KUKA KRL program: MyProgram_013().src

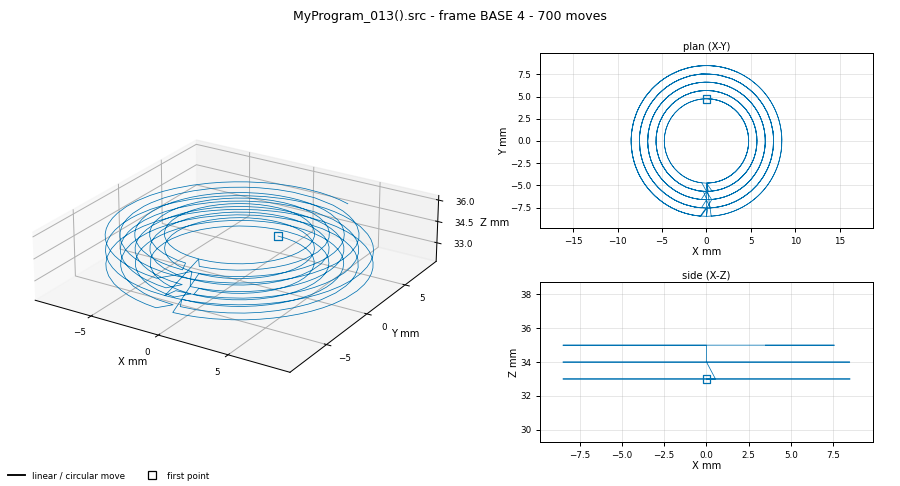
[picture p0: tool path of MyProgram_013().src in frame BASE 4, 700 of 700 moves have a stored position in this frame; points joined in program order, loops and branches not executed]
&ACCESS RVP
&REL 1
&PARAM TEMPLATE = C:\KRC\Roboter\Template\vorgabe
&PARAM EDITMASK = *
DEF MyProgram_013()
; ---- Setting reference (Base) ----
$BASE = BASE_DATA[4]

; --------------------------
; ---- Setting tool (TCP) ----
$TOOL = TOOL_DATA[3]
; --------------------------

$VEL.CP = VEL_APROX_PRINT
Startdeposition()
$VEL.CP = VEL_PRINT
LIN {X -0.0007,Y 4.7501,Z 33,A -2.5066,B 0,C 0,E1 0.1598,E2 90.0722} C_DIS
LIN {X 0.6681,Y 4.7058,Z 33,A -2.4838,B 0,C 0,E1 0.1598,E2 90.0722} C_DIS
LIN {X 1.3234,Y 4.564,Z 33,A -2.4657,B 0,C 0,E1 0.1598,E2 90.0722} C_DIS
LIN {X 1.9517,Y 4.3306,Z 33,A -2.4524,B 0,C 0,E1 0.1598,E2 90.0722} C_DIS
LIN {X 2.5415,Y 4.0125,Z 33,A -2.4441,B 0,C 0,E1 0.1598,E2 90.0722} C_DIS
LIN {X 3.0824,Y 3.6166,Z 33,A -2.441,B 0,C 0,E1 0.1598,E2 90.0722} C_DIS
LIN {X 3.561,Y 3.1471,Z 33,A -2.4432,B 0,C 0,E1 0.1598,E2 90.0722} C_DIS
LIN {X 3.9664,Y 2.6132,Z 33,A -2.4509,B 0,C 0,E1 0.1598,E2 90.0722} C_DIS
LIN {X 4.2946,Y 2.0289,Z 33,A -2.4637,B 0,C 0,E1 0.1598,E2 90.0721} C_DIS
LIN {X 4.5387,Y 1.4047,Z 33,A -2.4812,B 0,C 0,E1 0.1598,E2 90.0721} C_DIS
LIN {X 4.6913,Y 0.7521,Z 33,A -2.5033,B 0,C 0,E1 0.1598,E2 90.072} C_DIS
LIN {X 4.7501,Y 0.0845,Z 33,A -2.5295,B 0,C 0,E1 0.1598,E2 90.072} C_DIS
LIN {X 4.7153,Y -0.5848,Z 33,A -2.5593,B 0,C 0,E1 0.1598,E2 90.072} C_DIS
LIN {X 4.5852,Y -1.2423,Z 33,A -2.592,B 0,C 0,E1 0.1598,E2 90.0719} C_DIS
LIN {X 4.3645,Y -1.8751,Z 33,A -2.6271,B 0,C 0,E1 0.1598,E2 90.0719} C_DIS
LIN {X 4.0581,Y -2.4712,Z 33,A -2.6637,B 0,C 0,E1 0.1598,E2 90.0719} C_DIS
LIN {X 3.6691,Y -3.0171,Z 33,A -2.7013,B 0,C 0,E1 0.1598,E2 90.0719} C_DIS
LIN {X 3.2075,Y -3.5028,Z 33,A -2.7389,B 0,C 0,E1 0.1598,E2 90.0719} C_DIS
LIN {X 2.6831,Y -3.9201,Z 33,A -2.776,B 0,C 0,E1 0.1598,E2 90.0718} C_DIS
LIN {X 2.1055,Y -4.2604,Z 33,A -2.8117,B 0,C 0,E1 0.1598,E2 90.0718} C_DIS
LIN {X 1.4851,Y -4.5147,Z 33,A -2.8453,B 0,C 0,E1 0.1598,E2 90.0718} C_DIS
LIN {X 0.8351,Y -4.6789,Z 33,A -2.8762,B 0,C 0,E1 0.1598,E2 90.0718} C_DIS
LIN {X 0.0007,Y -4.7531,Z 33,A -2.9099,B 0,C 0,E1 0.1598,E2 90.0717} C_DIS
Enddeposition()
LIN {X 0.0007,Y -4.7531,Z 33,A -2.9099,B 0,C 0,E1 0.1598,E2 90.0717} C_DIS
Startdeposition()
$VEL.CP = VEL_PRINT
LIN {X 0.2137,Y -5.6787,Z 33,A -2.941,B 0,C 0,E1 0.1598,E2 90.0711} C_DIS
LIN {X 1.0439,Y -5.585,Z 33,A -2.9071,B 0,C 0,E1 0.1598,E2 90.0717} C_DIS
LIN {X 1.8527,Y -5.375,Z 33,A -2.8685,B 0,C 0,E1 0.1598,E2 90.0717} C_DIS
LIN {X 2.6206,Y -5.0447,Z 33,A -2.8262,B 0,C 0,E1 0.1598,E2 90.0717} C_DIS
LIN {X 3.3323,Y -4.6064,Z 33,A -2.7814,B 0,C 0,E1 0.1598,E2 90.0717} C_DIS
LIN {X 3.9709,Y -4.067,Z 33,A -2.735,B 0,C 0,E1 0.1598,E2 90.0717} C_DIS
LIN {X 4.5249,Y -3.4414,Z 33,A -2.6879,B 0,C 0,E1 0.1598,E2 90.0717} C_DIS
LIN {X 4.9785,Y -2.7397,Z 33,A -2.6413,B 0,C 0,E1 0.1598,E2 90.0717} C_DIS
LIN {X 5.3268,Y -1.9802,Z 33,A -2.5962,B 0,C 0,E1 0.1598,E2 90.0717} C_DIS
LIN {X 5.5609,Y -1.178,Z 33,A -2.5534,B 0,C 0,E1 0.1598,E2 90.0718} C_DIS
LIN {X 5.6744,Y -0.3499,Z 33,A -2.5139,B 0,C 0,E1 0.1598,E2 90.0718} C_DIS
LIN {X 5.6653,Y 0.4859,Z 33,A -2.4786,B 0,C 0,E1 0.1598,E2 90.0718} C_DIS
LIN {X 5.5351,Y 1.3214,Z 33,A -2.4477,B 0,C 0,E1 0.1598,E2 90.0717} C_DIS
LIN {X 5.3036,Y 2.0495,Z 33,A -2.4255,B 0,C 0,E1 0.1598,E2 90.072} C_DIS
LIN {X 4.9443,Y 2.804,Z 33,A -2.4066,B 0,C 0,E1 0.1598,E2 90.072} C_DIS
LIN {X 4.4801,Y 3.4987,Z 33,A -2.3942,B 0,C 0,E1 0.1598,E2 90.072} C_DIS
LIN {X 3.919,Y 4.1181,Z 33,A -2.3887,B 0,C 0,E1 0.1598,E2 90.0722} C_DIS
LIN {X 3.2725,Y 4.6475,Z 33,A -2.3901,B 0,C 0,E1 0.1598,E2 90.0722} C_DIS
LIN {X 2.5558,Y 5.077,Z 33,A -2.3983,B 0,C 0,E1 0.1598,E2 90.0722} C_DIS
LIN {X 1.7838,Y 5.3965,Z 33,A -2.4133,B 0,C 0,E1 0.1598,E2 90.0722} C_DIS
LIN {X 0.9734,Y 5.6004,Z 33,A -2.4345,B 0,C 0,E1 0.1598,E2 90.0722} C_DIS
LIN {X 0.1419,Y 5.6813,Z 33,A -2.4618,B 0,C 0,E1 0.1598,E2 90.0722} C_DIS
LIN {X -0.6925,Y 5.6406,Z 33,A -2.4943,B 0,C 0,E1 0.1598,E2 90.0722} C_DIS
LIN {X -1.512,Y 5.4783,Z 33,A -2.5314,B 0,C 0,E1 0.1598,E2 90.0722} C_DIS
LIN {X -2.2998,Y 5.1998,Z 33,A -2.5722,B 0,C 0,E1 0.1598,E2 90.0722} C_DIS
LIN {X -3.0374,Y 4.8067,Z 33,A -2.616,B 0,C 0,E1 0.1598,E2 90.072} C_DIS
LIN {X -3.7082,Y 4.3081,Z 33,A -2.6618,B 0,C 0,E1 0.1598,E2 90.0719} C_DIS
LIN {X -4.3,Y 3.7181,Z 33,A -2.7085,B 0,C 0,E1 0.1598,E2 90.0718} C_DIS
LIN {X -4.7979,Y 3.0471,Z 33,A -2.7551,B 0,C 0,E1 0.1598,E2 90.0717} C_DIS
LIN {X -5.1942,Y 2.3114,Z 33,A -2.8008,B 0,C 0,E1 0.1598,E2 90.0716} C_DIS
LIN {X -5.4756,Y 1.5246,Z 33,A -2.8443,B 0,C 0,E1 0.1598,E2 90.0715} C_DIS
LIN {X -5.642,Y 0.7055,Z 33,A -2.8851,B 0,C 0,E1 0.1598,E2 90.0714} C_DIS
LIN {X -5.6824,Y -0.1291,Z 33,A -2.9218,B 0,C 0,E1 0.1598,E2 90.0714} C_DIS
LIN {X -5.6024,Y -0.9608,Z 33,A -2.9541,B 0,C 0,E1 0.1598,E2 90.0713} C_DIS
LIN {X -5.4025,Y -1.7721,Z 33,A -2.9811,B 0,C 0,E1 0.1598,E2 90.0713} C_DIS
LIN {X -5.0843,Y -2.545,Z 33,A -3.0021,B 0,C 0,E1 0.1598,E2 90.0713} C_DIS
LIN {X -4.3348,Y -3.6846,Z 33,A -3.0224,B 0,C 0,E1 0.1598,E2 90.0708} C_DIS
LIN {X -3.5478,Y -4.442,Z 33,A -3.026,B 0,C 0,E1 0.1598,E2 90.0712} C_DIS
LIN {X -2.9488,Y -4.8595,Z 33,A -3.0219,B 0,C 0,E1 0.1598,E2 90.0714} C_DIS
LIN {X -2.3018,Y -5.1977,Z 33,A -3.0126,B 0,C 0,E1 0.1598,E2 90.0714} C_DIS
LIN {X -1.6166,Y -5.4502,Z 33,A -2.9982,B 0,C 0,E1 0.1598,E2 90.0715} C_DIS
LIN {X -0.9048,Y -5.6125,Z 33,A -2.979,B 0,C 0,E1 0.1598,E2 90.0715} C_DIS
LIN {X 0.0047,Y -5.6869,Z 33,A -2.9488,B 0,C 0,E1 0.1598,E2 90.0716} C_DIS
Enddeposition()
LIN {X 0.0047,Y -5.6869,Z 33,A -2.9488,B 0,C 0,E1 0.1598,E2 90.0716} C_DIS
Startdeposition()
$VEL.CP = VEL_PRINT
LIN {X -0.594,Y -6.5924,Z 33,A -3.0088,B 0,C 0,E1 0.1598,E2 90.071} C_DIS
LIN {X -1.3414,Y -6.4806,Z 33,A -3.032,B 0,C 0,E1 0.1598,E2 90.0715} C_DIS
LIN {X -2.0715,Y -6.2858,Z 33,A -3.0505,B 0,C 0,E1 0.1598,E2 90.0715} C_DIS
LIN {X -2.7752,Y -6.0102,Z 33,A -3.0646,B 0,C 0,E1 0.1598,E2 90.0715} C_DIS
LIN {X -3.4428,Y -5.6559,Z 33,A -3.074,B 0,C 0,E1 0.1598,E2 90.0715} C_DIS
LIN {X -4.0637,Y -5.2249,Z 33,A -3.0785,B 0,C 0,E1 0.1598,E2 90.0714} C_DIS
LIN {X -4.6336,Y -4.7287,Z 33,A -3.0784,B 0,C 0,E1 0.1598,E2 90.0714} C_DIS
LIN {X -5.1419,Y -4.1694,Z 33,A -3.0733,B 0,C 0,E1 0.1598,E2 90.0714} C_DIS
LIN {X -5.584,Y -3.5562,Z 33,A -3.0636,B 0,C 0,E1 0.1598,E2 90.0713} C_DIS
LIN {X -5.9525,Y -2.8963,Z 33,A -3.0491,B 0,C 0,E1 0.1598,E2 90.0713} C_DIS
LIN {X -6.2423,Y -2.1982,Z 33,A -3.0302,B 0,C 0,E1 0.1598,E2 90.0713} C_DIS
LIN {X -6.4539,Y -1.4727,Z 33,A -3.0073,B 0,C 0,E1 0.1598,E2 90.0713} C_DIS
LIN {X -6.5775,Y -0.7272,Z 33,A -2.9803,B 0,C 0,E1 0.1598,E2 90.0713} C_DIS
LIN {X -6.6199,Y 0.0273,Z 33,A -2.9499,B 0,C 0,E1 0.1598,E2 90.0713} C_DIS
LIN {X -6.5728,Y 0.7816,Z 33,A -2.9163,B 0,C 0,E1 0.1598,E2 90.0713} C_DIS
LIN {X -6.4409,Y 1.5258,Z 33,A -2.88,B 0,C 0,E1 0.1598,E2 90.0714} C_DIS
LIN {X -6.2234,Y 2.2495,Z 33,A -2.8414,B 0,C 0,E1 0.1598,E2 90.0715} C_DIS
LIN {X -5.9271,Y 2.9446,Z 33,A -2.8012,B 0,C 0,E1 0.1598,E2 90.0715} C_DIS
LIN {X -5.5534,Y 3.6016,Z 33,A -2.7597,B 0,C 0,E1 0.1598,E2 90.0717} C_DIS
LIN {X -5.1068,Y 4.2114,Z 33,A -2.7175,B 0,C 0,E1 0.1598,E2 90.0717} C_DIS
LIN {X -4.593,Y 4.7654,Z 33,A -2.6752,B 0,C 0,E1 0.1598,E2 90.0719} C_DIS
LIN {X -4.0195,Y 5.2576,Z 33,A -2.6332,B 0,C 0,E1 0.1598,E2 90.0719} C_DIS
LIN {X -3.3938,Y 5.6812,Z 33,A -2.5923,B 0,C 0,E1 0.1598,E2 90.072} C_DIS
LIN {X -2.7242,Y 6.0315,Z 33,A -2.5528,B 0,C 0,E1 0.1598,E2 90.0721} C_DIS
LIN {X -2.0191,Y 6.3032,Z 33,A -2.5153,B 0,C 0,E1 0.1598,E2 90.0721} C_DIS
LIN {X -1.2873,Y 6.4926,Z 33,A -2.4803,B 0,C 0,E1 0.1598,E2 90.0722} C_DIS
LIN {X -0.5389,Y 6.5981,Z 33,A -2.4483,B 0,C 0,E1 0.1598,E2 90.0723} C_DIS
LIN {X 0.2166,Y 6.6144,Z 33,A -2.4197,B 0,C 0,E1 0.1598,E2 90.0723} C_DIS
LIN {X 0.9691,Y 6.5467,Z 33,A -2.3948,B 0,C 0,E1 0.1598,E2 90.0723} C_DIS
LIN {X 1.7092,Y 6.3938,Z 33,A -2.3739,B 0,C 0,E1 0.1598,E2 90.0723} C_DIS
LIN {X 2.427,Y 6.1575,Z 33,A -2.3575,B 0,C 0,E1 0.1598,E2 90.0723} C_DIS
LIN {X 3.1139,Y 5.8421,Z 33,A -2.3455,B 0,C 0,E1 0.1598,E2 90.0723} C_DIS
LIN {X 3.7582,Y 5.447,Z 33,A -2.3385,B 0,C 0,E1 0.1598,E2 90.0723} C_DIS
LIN {X 4.3559,Y 4.9846,Z 33,A -2.336,B 0,C 0,E1 0.1598,E2 90.0723} C_DIS
LIN {X 4.8953,Y 4.455,Z 33,A -2.3386,B 0,C 0,E1 0.1598,E2 90.0723} C_DIS
LIN {X 5.3719,Y 3.8683,Z 33,A -2.3459,B 0,C 0,E1 0.1598,E2 90.0723} C_DIS
LIN {X 5.7789,Y 3.2314,Z 33,A -2.358,B 0,C 0,E1 0.1598,E2 90.0722} C_DIS
LIN {X 6.1095,Y 2.5518,Z 33,A -2.3747,B 0,C 0,E1 0.1598,E2 90.0722} C_DIS
LIN {X 6.3596,Y 1.8384,Z 33,A -2.3958,B 0,C 0,E1 0.1598,E2 90.0721} C_DIS
LIN {X 6.5283,Y 1.1016,Z 33,A -2.421,B 0,C 0,E1 0.1598,E2 90.0721} C_DIS
LIN {X 6.6097,Y 0.3501,Z 33,A -2.4499,B 0,C 0,E1 0.1598,E2 90.072} C_DIS
LIN {X 6.6083,Y -0.4056,Z 33,A -2.4822,B 0,C 0,E1 0.1598,E2 90.072} C_DIS
LIN {X 6.5167,Y -1.1559,Z 33,A -2.5175,B 0,C 0,E1 0.1598,E2 90.072} C_DIS
LIN {X 6.3411,Y -1.8908,Z 33,A -2.5553,B 0,C 0,E1 0.1598,E2 90.0719} C_DIS
LIN {X 6.0864,Y -2.6023,Z 33,A -2.595,B 0,C 0,E1 0.1598,E2 90.0719} C_DIS
LIN {X 5.75,Y -3.2792,Z 33,A -2.6362,B 0,C 0,E1 0.1598,E2 90.0719} C_DIS
LIN {X 5.3387,Y -3.9133,Z 33,A -2.6783,B 0,C 0,E1 0.1598,E2 90.0718} C_DIS
LIN {X 4.8584,Y -4.4969,Z 33,A -2.7208,B 0,C 0,E1 0.1598,E2 90.0718} C_DIS
LIN {X 4.3154,Y -5.0226,Z 33,A -2.7632,B 0,C 0,E1 0.1598,E2 90.0718} C_DIS
LIN {X 3.7137,Y -5.48,Z 33,A -2.8048,B 0,C 0,E1 0.1598,E2 90.0718} C_DIS
LIN {X 3.064,Y -5.8662,Z 33,A -2.8451,B 0,C 0,E1 0.1598,E2 90.0718} C_DIS
LIN {X 2.3756,Y -6.1779,Z 33,A -2.8836,B 0,C 0,E1 0.1598,E2 90.0717} C_DIS
LIN {X 1.6557,Y -6.4077,Z 33,A -2.9198,B 0,C 0,E1 0.1598,E2 90.0717} C_DIS
LIN {X 0.9145,Y -6.5546,Z 33,A -2.9533,B 0,C 0,E1 0.1598,E2 90.0717} C_DIS
LIN {X -0.0276,Y -6.6228,Z 33,A -2.9907,B 0,C 0,E1 0.1598,E2 90.0716} C_DIS
Enddeposition()
LIN {X -0.0276,Y -6.6228,Z 33,A -2.9907,B 0,C 0,E1 0.1598,E2 90.0716} C_DIS
Startdeposition()
$VEL.CP = VEL_PRINT
LIN {X 0.4585,Y -7.5385,Z 33,A -3.0114,B 0,C 0,E1 0.1598,E2 90.071} C_DIS
LIN {X 1.4933,Y -7.408,Z 33,A -2.9685,B 0,C 0,E1 0.1598,E2 90.0716} C_DIS
LIN {X 2.4321,Y -7.1566,Z 33,A -2.9234,B 0,C 0,E1 0.1598,E2 90.0716} C_DIS
LIN {X 3.3695,Y -6.7602,Z 33,A -2.8721,B 0,C 0,E1 0.1598,E2 90.0716} C_DIS
LIN {X 4.2493,Y -6.2487,Z 33,A -2.818,B 0,C 0,E1 0.1598,E2 90.0716} C_DIS
LIN {X 5.0198,Y -5.6498,Z 33,A -2.7642,B 0,C 0,E1 0.1598,E2 90.0717} C_DIS
LIN {X 5.777,Y -4.8711,Z 33,A -2.7031,B 0,C 0,E1 0.1598,E2 90.0717} C_DIS
LIN {X 6.3764,Y -4.0561,Z 33,A -2.6462,B 0,C 0,E1 0.1598,E2 90.0717} C_DIS
LIN {X 6.8946,Y -3.0967,Z 33,A -2.5862,B 0,C 0,E1 0.1598,E2 90.0717} C_DIS
LIN {X 7.243,Y -2.1568,Z 33,A -2.5334,B 0,C 0,E1 0.1598,E2 90.0717} C_DIS
LIN {X 7.5107,Y -0.834,Z 33,A -2.4665,B 0,C 0,E1 0.1598,E2 90.0712} C_DIS
LIN {X 7.5444,Y 0.3645,Z 33,A -2.4144,B 0,C 0,E1 0.1598,E2 90.0714} C_DIS
LIN {X 7.4758,Y 1.1076,Z 33,A -2.3857,B 0,C 0,E1 0.1598,E2 90.0719} C_DIS
LIN {X 7.2589,Y 2.0845,Z 33,A -2.352,B 0,C 0,E1 0.1598,E2 90.0719} C_DIS
LIN {X 6.8556,Y 3.181,Z 33,A -2.32,B 0,C 0,E1 0.1598,E2 90.0718} C_DIS
LIN {X 6.2145,Y 4.2988,Z 33,A -2.296,B 0,C 0,E1 0.1598,E2 90.0718} C_DIS
LIN {X 5.5266,Y 5.1537,Z 33,A -2.2853,B 0,C 0,E1 0.1598,E2 90.0721} C_DIS
LIN {X 4.8072,Y 5.8266,Z 33,A -2.2834,B 0,C 0,E1 0.1598,E2 90.0723} C_DIS
LIN {X 4.0099,Y 6.4049,Z 33,A -2.2883,B 0,C 0,E1 0.1598,E2 90.0723} C_DIS
LIN {X 3.0731,Y 6.9046,Z 33,A -2.3017,B 0,C 0,E1 0.1598,E2 90.0723} C_DIS
LIN {X 1.8528,Y 7.3262,Z 33,A -2.3289,B 0,C 0,E1 0.1598,E2 90.0723} C_DIS
LIN {X 0.3601,Y 7.5484,Z 33,A -2.3747,B 0,C 0,E1 0.1598,E2 90.0723} C_DIS
LIN {X -0.7846,Y 7.5163,Z 33,A -2.4183,B 0,C 0,E1 0.1598,E2 90.0723} C_DIS
LIN {X -1.8547,Y 7.3257,Z 33,A -2.4659,B 0,C 0,E1 0.1598,E2 90.0723} C_DIS
LIN {X -3.0695,Y 6.9061,Z 33,A -2.5284,B 0,C 0,E1 0.1598,E2 90.0721} C_DIS
LIN {X -4.1555,Y 6.3135,Z 33,A -2.5934,B 0,C 0,E1 0.1598,E2 90.0719} C_DIS
LIN {X -4.9937,Y 5.6676,Z 33,A -2.6516,B 0,C 0,E1 0.1598,E2 90.0719} C_DIS
LIN {X -5.8601,Y 4.7735,Z 33,A -2.7211,B 0,C 0,E1 0.1598,E2 90.0715} C_DIS
LIN {X -6.5519,Y 3.7675,Z 33,A -2.789,B 0,C 0,E1 0.1598,E2 90.0714} C_DIS
LIN {X -7.0322,Y 2.7554,Z 33,A -2.8494,B 0,C 0,E1 0.1598,E2 90.0713} C_DIS
LIN {X -7.3835,Y 1.61,Z 33,A -2.9106,B 0,C 0,E1 0.1598,E2 90.0711} C_DIS
LIN {X -7.5294,Y 0.6625,Z 33,A -2.9561,B 0,C 0,E1 0.1598,E2 90.0711} C_DIS
LIN {X -7.555,Y -0.1736,Z 33,A -2.9925,B 0,C 0,E1 0.1598,E2 90.0712} C_DIS
LIN {X -7.4385,Y -1.3116,Z 33,A -3.0359,B 0,C 0,E1 0.1598,E2 90.0708} C_DIS
LIN {X -7.1813,Y -2.3543,Z 33,A -3.0706,B 0,C 0,E1 0.1598,E2 90.0708} C_DIS
LIN {X -6.7678,Y -3.3531,Z 33,A -3.0978,B 0,C 0,E1 0.1598,E2 90.0709} C_DIS
LIN {X -6.4075,Y -3.9965,Z 33,A -3.1121,B 0,C 0,E1 0.1598,E2 90.0712} C_DIS
LIN {X -5.9875,Y -4.6024,Z 33,A -3.1223,B 0,C 0,E1 0.1598,E2 90.0712} C_DIS
LIN {X -5.5098,Y -5.1641,Z 33,A -3.1286,B 0,C 0,E1 0.1598,E2 90.0712} C_DIS
LIN {X -4.7184,Y -5.9038,Z 33,A -3.1308,B 0,C 0,E1 0.1598,E2 90.0712} C_DIS
LIN {X -3.6178,Y -6.6342,Z 33,A -3.1214,B 0,C 0,E1 0.1598,E2 90.0712} C_DIS
LIN {X -2.4866,Y -7.1322,Z 33,A -3.1012,B 0,C 0,E1 0.1598,E2 90.0712} C_DIS
LIN {X -1.3594,Y -7.4352,Z 33,A -3.0728,B 0,C 0,E1 0.1598,E2 90.0714} C_DIS
LIN {X -0.0504,Y -7.555,Z 33,A -3.0299,B 0,C 0,E1 0.1598,E2 90.0715} C_DIS
Enddeposition()
LIN {X -0.0504,Y -7.555,Z 33,A -3.0299,B 0,C 0,E1 0.1598,E2 90.0715} C_DIS
Startdeposition()
$VEL.CP = VEL_PRINT
LIN {X -0.7006,Y -8.4584,Z 33,A -3.0918,B 0,C 0,E1 0.1598,E2 90.0709} C_DIS
LIN {X -1.5422,Y -8.3453,Z 33,A -3.1184,B 0,C 0,E1 0.1598,E2 90.0714} C_DIS
LIN {X -2.3683,Y -8.149,Z 33,A -3.1403,B 0,C 0,E1 0.1598,E2 90.0714} C_DIS
LIN {X -3.1708,Y -7.8715,Z 33,A -3.1579,B 0,C 0,E1 0.1598,E2 90.0714} C_DIS
LIN {X -3.9414,Y -7.5148,Z 33,A -3.171,B 0,C 0,E1 0.1598,E2 90.0713} C_DIS
LIN {X -4.8509,Y -6.9678,Z 33,A -3.181,B 0,C 0,E1 0.1598,E2 90.0711} C_DIS
LIN {X -5.8026,Y -6.1979,Z 33,A -3.1832,B 0,C 0,E1 0.1598,E2 90.0711} C_DIS
LIN {X -6.5289,Y -5.4238,Z 33,A -3.1771,B 0,C 0,E1 0.1598,E2 90.0711} C_DIS
LIN {X -7.0385,Y -4.7444,Z 33,A -3.1671,B 0,C 0,E1 0.1598,E2 90.0711} C_DIS
LIN {X -7.5782,Y -3.8303,Z 33,A -3.148,B 0,C 0,E1 0.1598,E2 90.0709} C_DIS
LIN {X -8.0655,Y -2.6547,Z 33,A -3.116,B 0,C 0,E1 0.1598,E2 90.0707} C_DIS
LIN {X -8.3298,Y -1.6311,Z 33,A -3.0826,B 0,C 0,E1 0.1598,E2 90.071} C_DIS
LIN {X -8.4504,Y -0.794,Z 33,A -3.0518,B 0,C 0,E1 0.1598,E2 90.0711} C_DIS
LIN {X -8.4868,Y 0.2625,Z 33,A -3.0082,B 0,C 0,E1 0.1598,E2 90.0709} C_DIS
LIN {X -8.3733,Y 1.4065,Z 33,A -2.9558,B 0,C 0,E1 0.1598,E2 90.0709} C_DIS
LIN {X -8.108,Y 2.5188,Z 33,A -2.899,B 0,C 0,E1 0.1598,E2 90.0711} C_DIS
LIN {X -7.7027,Y 3.5617,Z 33,A -2.8402,B 0,C 0,E1 0.1598,E2 90.0713} C_DIS
LIN {X -7.171,Y 4.5462,Z 33,A -2.779,B 0,C 0,E1 0.1598,E2 90.0713} C_DIS
LIN {X -6.4514,Y 5.5151,Z 33,A -2.7116,B 0,C 0,E1 0.1598,E2 90.0714} C_DIS
LIN {X -5.8412,Y 6.1564,Z 33,A -2.6623,B 0,C 0,E1 0.1598,E2 90.0718} C_DIS
LIN {X -5.1684,Y 6.7318,Z 33,A -2.6133,B 0,C 0,E1 0.1598,E2 90.0719} C_DIS
LIN {X -4.4395,Y 7.2341,Z 33,A -2.5652,B 0,C 0,E1 0.1598,E2 90.072} C_DIS
LIN {X -3.4624,Y 7.7536,Z 33,A -2.5072,B 0,C 0,E1 0.1598,E2 90.072} C_DIS
LIN {X -2.342,Y 8.1581,Z 33,A -2.4488,B 0,C 0,E1 0.1598,E2 90.0722} C_DIS
LIN {X -1.6347,Y 8.3322,Z 33,A -2.4153,B 0,C 0,E1 0.1598,E2 90.0723} C_DIS
LIN {X -0.4279,Y 8.4768,Z 33,A -2.3647,B 0,C 0,E1 0.1598,E2 90.0724} C_DIS
LIN {X 0.3753,Y 8.4839,Z 33,A -2.3347,B 0,C 0,E1 0.1598,E2 90.0724} C_DIS
LIN {X 1.4195,Y 8.3683,Z 33,A -2.301,B 0,C 0,E1 0.1598,E2 90.0724} C_DIS
LIN {X 2.4431,Y 8.1317,Z 33,A -2.2732,B 0,C 0,E1 0.1598,E2 90.0724} C_DIS
LIN {X 3.5076,Y 7.7288,Z 33,A -2.2509,B 0,C 0,E1 0.1598,E2 90.0724} C_DIS
LIN {X 4.2643,Y 7.3384,Z 33,A -2.2396,B 0,C 0,E1 0.1598,E2 90.0724} C_DIS
LIN {X 4.978,Y 6.8742,Z 33,A -2.2329,B 0,C 0,E1 0.1598,E2 90.0724} C_DIS
LIN {X 5.6418,Y 6.3409,Z 33,A -2.2311,B 0,C 0,E1 0.1598,E2 90.0724} C_DIS
LIN {X 6.2488,Y 5.7439,Z 33,A -2.234,B 0,C 0,E1 0.1598,E2 90.0724} C_DIS
LIN {X 6.7931,Y 5.0892,Z 33,A -2.2417,B 0,C 0,E1 0.1598,E2 90.0724} C_DIS
LIN {X 7.2685,Y 4.3829,Z 33,A -2.2542,B 0,C 0,E1 0.1598,E2 90.0723} C_DIS
LIN {X 7.6714,Y 3.633,Z 33,A -2.2713,B 0,C 0,E1 0.1598,E2 90.0723} C_DIS
LIN {X 7.9967,Y 2.8463,Z 33,A -2.2927,B 0,C 0,E1 0.1598,E2 90.0721} C_DIS
LIN {X 8.2412,Y 2.0308,Z 33,A -2.3184,B 0,C 0,E1 0.1598,E2 90.0721} C_DIS
LIN {X 8.403,Y 1.1949,Z 33,A -2.3481,B 0,C 0,E1 0.1598,E2 90.0721} C_DIS
LIN {X 8.4897,Y 0.1343,Z 33,A -2.3898,B 0,C 0,E1 0.1598,E2 90.0716} C_DIS
LIN {X 8.4111,Y -1.1705,Z 33,A -2.448,B 0,C 0,E1 0.1598,E2 90.0713} C_DIS
LIN {X 8.1697,Y -2.3009,Z 33,A -2.5053,B 0,C 0,E1 0.1598,E2 90.0715} C_DIS
LIN {X 7.902,Y -3.097,Z 33,A -2.5495,B 0,C 0,E1 0.1598,E2 90.0718} C_DIS
LIN {X 7.5569,Y -3.8628,Z 33,A -2.5949,B 0,C 0,E1 0.1598,E2 90.0718} C_DIS
LIN {X 7.1379,Y -4.5907,Z 33,A -2.6413,B 0,C 0,E1 0.1598,E2 90.0718} C_DIS
LIN {X 6.6491,Y -5.2737,Z 33,A -2.6884,B 0,C 0,E1 0.1598,E2 90.0718} C_DIS
LIN {X 6.0952,Y -5.9051,Z 33,A -2.7357,B 0,C 0,E1 0.1598,E2 90.0718} C_DIS
LIN {X 5.4818,Y -6.4787,Z 33,A -2.7827,B 0,C 0,E1 0.1598,E2 90.0717} C_DIS
LIN {X 4.8147,Y -6.9889,Z 33,A -2.8289,B 0,C 0,E1 0.1598,E2 90.0717} C_DIS
LIN {X 4.1004,Y -7.4306,Z 33,A -2.874,B 0,C 0,E1 0.1598,E2 90.0717} C_DIS
LIN {X 3.043,Y -7.927,Z 33,A -2.9339,B 0,C 0,E1 0.1598,E2 90.0716} C_DIS
LIN {X 2.0967,Y -8.224,Z 33,A -2.9812,B 0,C 0,E1 0.1598,E2 90.0716} C_DIS
LIN {X 1.3193,Y -8.3829,Z 33,A -3.0165,B 0,C 0,E1 0.1598,E2 90.0716} C_DIS
LIN {X 0.5306,Y -8.4691,Z 33,A -3.0491,B 0,C 0,E1 0.1598,E2 90.0716} C_DIS
LIN {X 0.5306,Y -8.4691,Z 33,A -3.0491,B 0,C 0,E1 0.1598,E2 90.0716} C_DIS
Enddeposition()
LIN {X 0.0007,Y -4.7532,Z 34,A -2.8958,B 0,C 0,E1 0.1598,E2 90.0604} C_DIS
Startdeposition()
$VEL.CP = VEL_PRINT
LIN {X 0.0007,Y -4.7532,Z 34,A -2.9015,B 0,C 0,E1 0.1598,E2 90.0661} C_DIS
LIN {X 0.9486,Y -4.6542,Z 34,A -2.8674,B 0,C 0,E1 0.1598,E2 90.0711} C_DIS
LIN {X 1.616,Y -4.4661,Z 34,A -2.8355,B 0,C 0,E1 0.1598,E2 90.0717} C_DIS
LIN {X 2.1728,Y -4.2245,Z 34,A -2.8048,B 0,C 0,E1 0.1598,E2 90.0718} C_DIS
LIN {X 2.7642,Y -3.8623,Z 34,A -2.7676,B 0,C 0,E1 0.1598,E2 90.0718} C_DIS
LIN {X 3.2975,Y -3.419,Z 34,A -2.7292,B 0,C 0,E1 0.1598,E2 90.0718} C_DIS
LIN {X 3.7622,Y -2.904,Z 34,A -2.6901,B 0,C 0,E1 0.1598,E2 90.0718} C_DIS
LIN {X 4.1442,Y -2.3248,Z 34,A -2.6514,B 0,C 0,E1 0.1598,E2 90.0718} C_DIS
LIN {X 4.4373,Y -1.6963,Z 34,A -2.6139,B 0,C 0,E1 0.1598,E2 90.0718} C_DIS
LIN {X 4.6365,Y -1.032,Z 34,A -2.5782,B 0,C 0,E1 0.1598,E2 90.0718} C_DIS
LIN {X 4.739,Y -0.346,Z 34,A -2.5453,B 0,C 0,E1 0.1598,E2 90.0719} C_DIS
LIN {X 4.7366,Y 0.3475,Z 34,A -2.5158,B 0,C 0,E1 0.1598,E2 90.0719} C_DIS
LIN {X 4.6356,Y 1.0334,Z 34,A -2.4904,B 0,C 0,E1 0.1598,E2 90.0719} C_DIS
LIN {X 4.4387,Y 1.6985,Z 34,A -2.4693,B 0,C 0,E1 0.1598,E2 90.072} C_DIS
LIN {X 4.1427,Y 2.3258,Z 34,A -2.4536,B 0,C 0,E1 0.1598,E2 90.072} C_DIS
LIN {X 3.7591,Y 2.9036,Z 34,A -2.4432,B 0,C 0,E1 0.1598,E2 90.0721} C_DIS
LIN {X 3.2966,Y 3.4205,Z 34,A -2.4383,B 0,C 0,E1 0.1598,E2 90.0721} C_DIS
LIN {X 2.6918,Y 3.9131,Z 34,A -2.4397,B 0,C 0,E1 0.1598,E2 90.0721} C_DIS
LIN {X 2.1716,Y 4.2257,Z 34,A -2.4457,B 0,C 0,E1 0.1598,E2 90.0722} C_DIS
LIN {X 1.5337,Y 4.4982,Z 34,A -2.4576,B 0,C 0,E1 0.1598,E2 90.0722} C_DIS
LIN {X 0.8625,Y 4.6738,Z 34,A -2.4749,B 0,C 0,E1 0.1598,E2 90.0722} C_DIS
LIN {X 0.1729,Y 4.7478,Z 34,A -2.4972,B 0,C 0,E1 0.1598,E2 90.0722} C_DIS
LIN {X -0.5203,Y 4.7226,Z 34,A -2.5239,B 0,C 0,E1 0.1598,E2 90.0722} C_DIS
LIN {X -1.2022,Y 4.5961,Z 34,A -2.5544,B 0,C 0,E1 0.1598,E2 90.0722} C_DIS
LIN {X -1.9377,Y 4.3361,Z 34,A -2.5925,B 0,C 0,E1 0.1598,E2 90.0721} C_DIS
LIN {X -2.4755,Y 4.0551,Z 34,A -2.6242,B 0,C 0,E1 0.1598,E2 90.0721} C_DIS
LIN {X -3.0399,Y 3.6517,Z 34,A -2.662,B 0,C 0,E1 0.1598,E2 90.0719} C_DIS
LIN {X -3.5392,Y 3.1702,Z 34,A -2.7007,B 0,C 0,E1 0.1598,E2 90.0719} C_DIS
LIN {X -3.9639,Y 2.6216,Z 34,A -2.7395,B 0,C 0,E1 0.1598,E2 90.0718} C_DIS
LIN {X -4.3022,Y 2.016,Z 34,A -2.7776,B 0,C 0,E1 0.1598,E2 90.0717} C_DIS
LIN {X -4.5485,Y 1.3677,Z 34,A -2.8141,B 0,C 0,E1 0.1598,E2 90.0717} C_DIS
LIN {X -4.6999,Y 0.6909,Z 34,A -2.8483,B 0,C 0,E1 0.1598,E2 90.0716} C_DIS
LIN {X -4.7505,Y -0.0007,Z 34,A -2.8794,B 0,C 0,E1 0.1598,E2 90.0715} C_DIS
LIN {X -4.701,Y -0.6925,Z 34,A -2.9068,B 0,C 0,E1 0.1598,E2 90.0715} C_DIS
LIN {X -4.548,Y -1.369,Z 34,A -2.9298,B 0,C 0,E1 0.1598,E2 90.0715} C_DIS
LIN {X -4.2999,Y -2.0165,Z 34,A -2.9481,B 0,C 0,E1 0.1598,E2 90.0715} C_DIS
LIN {X -3.9613,Y -2.6217,Z 34,A -2.9614,B 0,C 0,E1 0.1598,E2 90.0715} C_DIS
LIN {X -3.5371,Y -3.1703,Z 34,A -2.9691,B 0,C 0,E1 0.1598,E2 90.0715} C_DIS
LIN {X -2.9701,Y -3.7059,Z 34,A -2.971,B 0,C 0,E1 0.1598,E2 90.0715} C_DIS
LIN {X -2.474,Y -4.0553,Z 34,A -2.9676,B 0,C 0,E1 0.1598,E2 90.0715} C_DIS
LIN {X -1.8569,Y -4.3718,Z 34,A -2.9584,B 0,C 0,E1 0.1598,E2 90.0715} C_DIS
LIN {X -1.2007,Y -4.5962,Z 34,A -2.9439,B 0,C 0,E1 0.1598,E2 90.0716} C_DIS
LIN {X -0.519,Y -4.7241,Z 34,A -2.9243,B 0,C 0,E1 0.1598,E2 90.0716} C_DIS
LIN {X -0.519,Y -4.7241,Z 34,A -2.9243,B 0,C 0,E1 0.1598,E2 90.0716} C_DIS
Enddeposition()
LIN {X 0.0049,Y -5.6869,Z 34,A -2.9449,B 0,C 0,E1 0.1598,E2 90.0705} C_DIS
Startdeposition()
$VEL.CP = VEL_PRINT
LIN {X -0.9378,Y -5.6119,Z 34,A -2.9774,B 0,C 0,E1 0.1598,E2 90.0715} C_DIS
LIN {X -2.248,Y -5.2264,Z 34,A -3.0091,B 0,C 0,E1 0.1598,E2 90.0715} C_DIS
LIN {X -3.1196,Y -4.7597,Z 34,A -3.0213,B 0,C 0,E1 0.1598,E2 90.0714} C_DIS
LIN {X -3.9338,Y -4.1051,Z 34,A -3.0233,B 0,C 0,E1 0.1598,E2 90.0714} C_DIS
LIN {X -4.4924,Y -3.4835,Z 34,A -3.0175,B 0,C 0,E1 0.1598,E2 90.0714} C_DIS
LIN {X -4.9545,Y -2.7873,Z 34,A -3.0049,B 0,C 0,E1 0.1598,E2 90.0714} C_DIS
LIN {X -5.3084,Y -2.0304,Z 34,A -2.9859,B 0,C 0,E1 0.1598,E2 90.0713} C_DIS
LIN {X -5.5491,Y -1.2304,Z 34,A -2.9608,B 0,C 0,E1 0.1598,E2 90.0713} C_DIS
LIN {X -5.671,Y -0.4036,Z 34,A -2.9303,B 0,C 0,E1 0.1598,E2 90.0713} C_DIS
LIN {X -5.6695,Y 0.4321,Z 34,A -2.8949,B 0,C 0,E1 0.1598,E2 90.0713} C_DIS
LIN {X -5.5441,Y 1.2584,Z 34,A -2.8553,B 0,C 0,E1 0.1598,E2 90.0714} C_DIS
LIN {X -5.2975,Y 2.0568,Z 34,A -2.8125,B 0,C 0,E1 0.1598,E2 90.0714} C_DIS
LIN {X -4.9401,Y 2.8119,Z 34,A -2.7674,B 0,C 0,E1 0.1598,E2 90.0716} C_DIS
LIN {X -4.4743,Y 3.5056,Z 34,A -2.721,B 0,C 0,E1 0.1598,E2 90.0716} C_DIS
LIN {X -3.9112,Y 4.1229,Z 34,A -2.6742,B 0,C 0,E1 0.1598,E2 90.0718} C_DIS
LIN {X -3.2646,Y 4.6518,Z 34,A -2.628,B 0,C 0,E1 0.1598,E2 90.0719} C_DIS
LIN {X -2.5472,Y 5.0801,Z 34,A -2.5835,B 0,C 0,E1 0.1598,E2 90.072} C_DIS
LIN {X -1.7758,Y 5.4008,Z 34,A -2.5415,B 0,C 0,E1 0.1598,E2 90.0721} C_DIS
LIN {X -0.9649,Y 5.6032,Z 34,A -2.5031,B 0,C 0,E1 0.1598,E2 90.0722} C_DIS
LIN {X -0.1331,Y 5.6824,Z 34,A -2.4691,B 0,C 0,E1 0.1598,E2 90.0722} C_DIS
LIN {X 0.7013,Y 5.6393,Z 34,A -2.4401,B 0,C 0,E1 0.1598,E2 90.0723} C_DIS
LIN {X 1.5201,Y 5.4747,Z 34,A -2.4169,B 0,C 0,E1 0.1598,E2 90.0723} C_DIS
LIN {X 2.3063,Y 5.1926,Z 34,A -2.3998,B 0,C 0,E1 0.1598,E2 90.0723} C_DIS
LIN {X 3.0426,Y 4.7982,Z 34,A -2.3894,B 0,C 0,E1 0.1598,E2 90.0723} C_DIS
LIN {X 3.7136,Y 4.3007,Z 34,A -2.3857,B 0,C 0,E1 0.1598,E2 90.0723} C_DIS
LIN {X 4.304,Y 3.7099,Z 34,A -2.389,B 0,C 0,E1 0.1598,E2 90.0722} C_DIS
LIN {X 4.8012,Y 3.0387,Z 34,A -2.3992,B 0,C 0,E1 0.1598,E2 90.0722} C_DIS
LIN {X 5.1966,Y 2.3028,Z 34,A -2.4158,B 0,C 0,E1 0.1598,E2 90.072} C_DIS
LIN {X 5.4238,Y 1.7182,Z 34,A -2.4325,B 0,C 0,E1 0.1598,E2 90.0721} C_DIS
LIN {X 5.6677,Y 0.5136,Z 34,A -2.474,B 0,C 0,E1 0.1598,E2 90.0714} C_DIS
LIN {X 5.6679,Y -0.5137,Z 34,A -2.518,B 0,C 0,E1 0.1598,E2 90.0716} C_DIS
LIN {X 5.4828,Y -1.4969,Z 34,A -2.5668,B 0,C 0,E1 0.1598,E2 90.0716} C_DIS
LIN {X 5.2185,Y -2.2522,Z 34,A -2.6089,B 0,C 0,E1 0.1598,E2 90.0718} C_DIS
LIN {X 4.8495,Y -2.9621,Z 34,A -2.6527,B 0,C 0,E1 0.1598,E2 90.0718} C_DIS
LIN {X 4.3865,Y -3.6146,Z 34,A -2.6975,B 0,C 0,E1 0.1598,E2 90.0718} C_DIS
LIN {X 3.834,Y -4.1934,Z 34,A -2.7425,B 0,C 0,E1 0.1598,E2 90.0718} C_DIS
LIN {X 3.2072,Y -4.6905,Z 34,A -2.7867,B 0,C 0,E1 0.1598,E2 90.0718} C_DIS
LIN {X 2.5174,Y -5.0962,Z 34,A -2.8293,B 0,C 0,E1 0.1598,E2 90.0718} C_DIS
LIN {X 1.7771,Y -5.4004,Z 34,A -2.8695,B 0,C 0,E1 0.1598,E2 90.0718} C_DIS
LIN {X 1.0006,Y -5.5941,Z 34,A -2.9062,B 0,C 0,E1 0.1598,E2 90.0717} C_DIS
LIN {X 0.0049,Y -5.6869,Z 34,A -2.9467,B 0,C 0,E1 0.1598,E2 90.0717} C_DIS
Enddeposition()
LIN {X 0.0049,Y -5.6869,Z 34,A -2.9467,B 0,C 0,E1 0.1598,E2 90.0717} C_DIS
Startdeposition()
$VEL.CP = VEL_PRINT
LIN {X 0.5777,Y -6.5955,Z 34,A -2.9639,B 0,C 0,E1 0.1598,E2 90.071} C_DIS
LIN {X 1.3238,Y -6.4846,Z 34,A -2.9324,B 0,C 0,E1 0.1598,E2 90.0716} C_DIS
LIN {X 2.0528,Y -6.2912,Z 34,A -2.8974,B 0,C 0,E1 0.1598,E2 90.0716} C_DIS
LIN {X 2.7556,Y -6.018,Z 34,A -2.86,B 0,C 0,E1 0.1598,E2 90.0717} C_DIS
LIN {X 3.4221,Y -5.6648,Z 34,A -2.8205,B 0,C 0,E1 0.1598,E2 90.0717} C_DIS
LIN {X 4.0466,Y -5.2416,Z 34,A -2.7795,B 0,C 0,E1 0.1598,E2 90.0717} C_DIS
LIN {X 4.6157,Y -4.7464,Z 34,A -2.7375,B 0,C 0,E1 0.1598,E2 90.0717} C_DIS
LIN {X 5.1242,Y -4.1894,Z 34,A -2.6951,B 0,C 0,E1 0.1598,E2 90.0718} C_DIS
LIN {X 5.5676,Y -3.5791,Z 34,A -2.6528,B 0,C 0,E1 0.1598,E2 90.0718} C_DIS
LIN {X 5.9399,Y -2.923,Z 34,A -2.6111,B 0,C 0,E1 0.1598,E2 90.0718} C_DIS
LIN {X 6.232,Y -2.2275,Z 34,A -2.5707,B 0,C 0,E1 0.1598,E2 90.0718} C_DIS
LIN {X 6.4447,Y -1.504,Z 34,A -2.532,B 0,C 0,E1 0.1598,E2 90.0719} C_DIS
LIN {X 6.5746,Y -0.761,Z 34,A -2.4956,B 0,C 0,E1 0.1598,E2 90.0719} C_DIS
LIN {X 6.6192,Y -0.0082,Z 34,A -2.4618,B 0,C 0,E1 0.1598,E2 90.0719} C_DIS
LIN {X 6.578,Y 0.7451,Z 34,A -2.4313,B 0,C 0,E1 0.1598,E2 90.072} C_DIS
LIN {X 6.4502,Y 1.4885,Z 34,A -2.4043,B 0,C 0,E1 0.1598,E2 90.072} C_DIS
LIN {X 6.2394,Y 2.2129,Z 34,A -2.3813,B 0,C 0,E1 0.1598,E2 90.072} C_DIS
LIN {X 5.9462,Y 2.9079,Z 34,A -2.3625,B 0,C 0,E1 0.1598,E2 90.0721} C_DIS
LIN {X 5.5772,Y 3.5657,Z 34,A -2.3481,B 0,C 0,E1 0.1598,E2 90.0721} C_DIS
LIN {X 5.1349,Y 4.1767,Z 34,A -2.3385,B 0,C 0,E1 0.1598,E2 90.0722} C_DIS
LIN {X 4.626,Y 4.7336,Z 34,A -2.3336,B 0,C 0,E1 0.1598,E2 90.0722} C_DIS
LIN {X 4.058,Y 5.23,Z 34,A -2.3335,B 0,C 0,E1 0.1598,E2 90.0723} C_DIS
LIN {X 3.4363,Y 5.6572,Z 34,A -2.3383,B 0,C 0,E1 0.1598,E2 90.0723} C_DIS
LIN {X 2.7698,Y 6.0105,Z 34,A -2.3479,B 0,C 0,E1 0.1598,E2 90.0723} C_DIS
LIN {X 2.0685,Y 6.2881,Z 34,A -2.3621,B 0,C 0,E1 0.1598,E2 90.0723} C_DIS
LIN {X 1.3394,Y 6.481,Z 34,A -2.3808,B 0,C 0,E1 0.1598,E2 90.0723} C_DIS
LIN {X 0.5934,Y 6.5917,Z 34,A -2.4036,B 0,C 0,E1 0.1598,E2 90.0723} C_DIS
LIN {X -0.1604,Y 6.6168,Z 34,A -2.4304,B 0,C 0,E1 0.1598,E2 90.0723} C_DIS
LIN {X -0.912,Y 6.5551,Z 34,A -2.4608,B 0,C 0,E1 0.1598,E2 90.0723} C_DIS
LIN {X -1.652,Y 6.4092,Z 34,A -2.4942,B 0,C 0,E1 0.1598,E2 90.0723} C_DIS
LIN {X -2.3701,Y 6.1785,Z 34,A -2.5305,B 0,C 0,E1 0.1598,E2 90.0722} C_DIS
LIN {X -3.058,Y 5.8695,Z 34,A -2.5689,B 0,C 0,E1 0.1598,E2 90.0722} C_DIS
LIN {X -3.7059,Y 5.4833,Z 34,A -2.6091,B 0,C 0,E1 0.1598,E2 90.072} C_DIS
LIN {X -4.3058,Y 5.026,Z 34,A -2.6505,B 0,C 0,E1 0.1598,E2 90.072} C_DIS
LIN {X -4.8507,Y 4.5045,Z 34,A -2.6926,B 0,C 0,E1 0.1598,E2 90.0718} C_DIS
LIN {X -5.3311,Y 3.923,Z 34,A -2.7348,B 0,C 0,E1 0.1598,E2 90.0718} C_DIS
LIN {X -5.7425,Y 3.2908,Z 34,A -2.7767,B 0,C 0,E1 0.1598,E2 90.0717} C_DIS
LIN {X -6.0789,Y 2.6157,Z 34,A -2.8176,B 0,C 0,E1 0.1598,E2 90.0716} C_DIS
LIN {X -6.3375,Y 1.9072,Z 34,A -2.857,B 0,C 0,E1 0.1598,E2 90.0716} C_DIS
LIN {X -6.5493,Y 0.9884,Z 34,A -2.9034,B 0,C 0,E1 0.1598,E2 90.0712} C_DIS
LIN {X -6.62,Y -0.0624,Z 34,A -2.9503,B 0,C 0,E1 0.1598,E2 90.071} C_DIS
LIN {X -6.5736,Y -0.7867,Z 34,A -2.9795,B 0,C 0,E1 0.1598,E2 90.0713} C_DIS
LIN {X -6.4459,Y -1.5013,Z 34,A -3.0051,B 0,C 0,E1 0.1598,E2 90.0713} C_DIS
LIN {X -6.2438,Y -2.1983,Z 34,A -3.0272,B 0,C 0,E1 0.1598,E2 90.0713} C_DIS
LIN {X -5.9653,Y -2.8684,Z 34,A -3.0453,B 0,C 0,E1 0.1598,E2 90.0713} C_DIS
LIN {X -5.614,Y -3.5035,Z 34,A -3.0593,B 0,C 0,E1 0.1598,E2 90.0713} C_DIS
LIN {X -5.1978,Y -4.0982,Z 34,A -3.0692,B 0,C 0,E1 0.1598,E2 90.0713} C_DIS
LIN {X -4.7185,Y -4.6433,Z 34,A -3.0747,B 0,C 0,E1 0.1598,E2 90.0713} C_DIS
LIN {X -4.1813,Y -5.1312,Z 34,A -3.0757,B 0,C 0,E1 0.1598,E2 90.0713} C_DIS
LIN {X -3.5951,Y -5.5593,Z 34,A -3.0724,B 0,C 0,E1 0.1598,E2 90.0713} C_DIS
LIN {X -2.9652,Y -5.9199,Z 34,A -3.0646,B 0,C 0,E1 0.1598,E2 90.0714} C_DIS
LIN {X -2.299,Y -6.2079,Z 34,A -3.0524,B 0,C 0,E1 0.1598,E2 90.0714} C_DIS
LIN {X -1.6051,Y -6.421,Z 34,A -3.036,B 0,C 0,E1 0.1598,E2 90.0714} C_DIS
LIN {X -0.8926,Y -6.5592,Z 34,A -3.0158,B 0,C 0,E1 0.1598,E2 90.0715} C_DIS
LIN {X 0.0124,Y -6.6207,Z 34,A -2.9852,B 0,C 0,E1 0.1598,E2 90.0715} C_DIS
Enddeposition()
LIN {X 0.0124,Y -6.6207,Z 34,A -2.9852,B 0,C 0,E1 0.1598,E2 90.0715} C_DIS
Startdeposition()
$VEL.CP = VEL_PRINT
LIN {X -0.5759,Y -7.5325,Z 34,A -3.0451,B 0,C 0,E1 0.1598,E2 90.0709} C_DIS
LIN {X -1.2817,Y -7.4478,Z 34,A -3.0679,B 0,C 0,E1 0.1598,E2 90.0714} C_DIS
LIN {X -2.3217,Y -7.189,Z 34,A -3.0951,B 0,C 0,E1 0.1598,E2 90.0714} C_DIS
LIN {X -3.0235,Y -6.9235,Z 34,A -3.1095,B 0,C 0,E1 0.1598,E2 90.0714} C_DIS
LIN {X -3.6944,Y -6.5874,Z 34,A -3.1199,B 0,C 0,E1 0.1598,E2 90.0714} C_DIS
LIN {X -4.3294,Y -6.1879,Z 34,A -3.1262,B 0,C 0,E1 0.1598,E2 90.0714} C_DIS
LIN {X -5.0669,Y -5.6086,Z 34,A -3.1286,B 0,C 0,E1 0.1598,E2 90.0712} C_DIS
LIN {X -5.8305,Y -4.8019,Z 34,A -3.1222,B 0,C 0,E1 0.1598,E2 90.071} C_DIS
LIN {X -6.3104,Y -4.1509,Z 34,A -3.1124,B 0,C 0,E1 0.1598,E2 90.0712} C_DIS
LIN {X -6.7176,Y -3.4521,Z 34,A -3.0978,B 0,C 0,E1 0.1598,E2 90.0712} C_DIS
LIN {X -7.0469,Y -2.7135,Z 34,A -3.0786,B 0,C 0,E1 0.1598,E2 90.0712} C_DIS
LIN {X -7.353,Y -1.75,Z 34,A -3.0488,B 0,C 0,E1 0.1598,E2 90.0709} C_DIS
LIN {X -7.4928,Y -0.9918,Z 34,A -3.0222,B 0,C 0,E1 0.1598,E2 90.0713} C_DIS
LIN {X -7.5499,Y 0.3578,Z 34,A -2.9665,B 0,C 0,E1 0.1598,E2 90.0706} C_DIS
LIN {X -7.4272,Y 1.4016,Z 34,A -2.9183,B 0,C 0,E1 0.1598,E2 90.0711} C_DIS
LIN {X -7.1706,Y 2.3883,Z 34,A -2.8673,B 0,C 0,E1 0.1598,E2 90.0712} C_DIS
LIN {X -6.8023,Y 3.2788,Z 34,A -2.8162,B 0,C 0,E1 0.1598,E2 90.0714} C_DIS
LIN {X -6.2564,Y 4.2382,Z 34,A -2.7555,B 0,C 0,E1 0.1598,E2 90.0714} C_DIS
LIN {X -5.4688,Y 5.2145,Z 34,A -2.6852,B 0,C 0,E1 0.1598,E2 90.0715} C_DIS
LIN {X -4.5789,Y 6.0112,Z 34,A -2.6189,B 0,C 0,E1 0.1598,E2 90.0718} C_DIS
LIN {X -3.6474,Y 6.6179,Z 34,A -2.559,B 0,C 0,E1 0.1598,E2 90.072} C_DIS
LIN {X -2.4084,Y 7.1591,Z 34,A -2.4904,B 0,C 0,E1 0.1598,E2 90.0721} C_DIS
LIN {X -1.6689,Y 7.3711,Z 34,A -2.4543,B 0,C 0,E1 0.1598,E2 90.0723} C_DIS
LIN {X -0.5224,Y 7.5388,Z 34,A -2.4049,B 0,C 0,E1 0.1598,E2 90.0723} C_DIS
LIN {X 1.1633,Y 7.4668,Z 34,A -2.3457,B 0,C 0,E1 0.1598,E2 90.0724} C_DIS
LIN {X 2.7967,Y 7.022,Z 34,A -2.3041,B 0,C 0,E1 0.1598,E2 90.0724} C_DIS
LIN {X 3.8322,Y 6.5147,Z 34,A -2.2875,B 0,C 0,E1 0.1598,E2 90.0724} C_DIS
LIN {X 4.5903,Y 5.996,Z 34,A -2.2815,B 0,C 0,E1 0.1598,E2 90.0724} C_DIS
LIN {X 5.152,Y 5.5223,Z 34,A -2.2809,B 0,C 0,E1 0.1598,E2 90.0724} C_DIS
LIN {X 5.7873,Y 4.8591,Z 34,A -2.2856,B 0,C 0,E1 0.1598,E2 90.0722} C_DIS
LIN {X 6.4119,Y 3.9934,Z 34,A -2.2992,B 0,C 0,E1 0.1598,E2 90.072} C_DIS
LIN {X 6.8539,Y 3.1845,Z 34,A -2.3173,B 0,C 0,E1 0.1598,E2 90.072} C_DIS
LIN {X 7.257,Y 2.1123,Z 34,A -2.3479,B 0,C 0,E1 0.1598,E2 90.0717} C_DIS
LIN {X 7.4816,Y 1.0715,Z 34,A -2.3841,B 0,C 0,E1 0.1598,E2 90.0718} C_DIS
LIN {X 7.555,Y 0.1719,Z 34,A -2.4198,B 0,C 0,E1 0.1598,E2 90.0719} C_DIS
LIN {X 7.4788,Y -1.0567,Z 34,A -2.4745,B 0,C 0,E1 0.1598,E2 90.0713} C_DIS
LIN {X 7.3337,Y -1.8239,Z 34,A -2.513,B 0,C 0,E1 0.1598,E2 90.0717} C_DIS
LIN {X 7.0562,Y -2.693,Z 34,A -2.5603,B 0,C 0,E1 0.1598,E2 90.0717} C_DIS
LIN {X 6.7642,Y -3.3619,Z 34,A -2.5997,B 0,C 0,E1 0.1598,E2 90.0719} C_DIS
LIN {X 6.3137,Y -4.1553,Z 34,A -2.6499,B 0,C 0,E1 0.1598,E2 90.0717} C_DIS
LIN {X 5.6885,Y -4.9745,Z 34,A -2.7078,B 0,C 0,E1 0.1598,E2 90.0717} C_DIS
LIN {X 5.0183,Y -5.6511,Z 34,A -2.7613,B 0,C 0,E1 0.1598,E2 90.0717} C_DIS
LIN {X 4.2052,Y -6.2792,Z 34,A -2.818,B 0,C 0,E1 0.1598,E2 90.0717} C_DIS
LIN {X 3.1862,Y -6.8483,Z 34,A -2.8796,B 0,C 0,E1 0.1598,E2 90.0716} C_DIS
LIN {X 2.2593,Y -7.211,Z 34,A -2.9291,B 0,C 0,E1 0.1598,E2 90.0716} C_DIS
LIN {X 1.2096,Y -7.4594,Z 34,A -2.9782,B 0,C 0,E1 0.1598,E2 90.0716} C_DIS
LIN {X 0.1546,Y -7.5554,Z 34,A -3.021,B 0,C 0,E1 0.1598,E2 90.0716} C_DIS
LIN {X 0.1546,Y -7.5554,Z 34,A -3.021,B 0,C 0,E1 0.1598,E2 90.0716} C_DIS
Enddeposition()
LIN {X -0.0093,Y -8.4875,Z 34,A -3.0657,B 0,C 0,E1 0.1598,E2 90.0703} C_DIS
Startdeposition()
$VEL.CP = VEL_PRINT
LIN {X 0.9615,Y -8.431,Z 34,A -3.0288,B 0,C 0,E1 0.1598,E2 90.0715} C_DIS
LIN {X 1.7297,Y -8.3081,Z 34,A -2.9955,B 0,C 0,E1 0.1598,E2 90.0715} C_DIS
LIN {X 2.4837,Y -8.1159,Z 34,A -2.9596,B 0,C 0,E1 0.1598,E2 90.0716} C_DIS
LIN {X 3.5402,Y -7.719,Z 34,A -2.904,B 0,C 0,E1 0.1598,E2 90.0716} C_DIS
LIN {X 4.4628,Y -7.2186,Z 34,A -2.8488,B 0,C 0,E1 0.1598,E2 90.0716} C_DIS
LIN {X 5.1543,Y -6.7421,Z 34,A -2.8031,B 0,C 0,E1 0.1598,E2 90.0717} C_DIS
LIN {X 5.7953,Y -6.1997,Z 34,A -2.7564,B 0,C 0,E1 0.1598,E2 90.0717} C_DIS
LIN {X 6.3796,Y -5.5965,Z 34,A -2.7092,B 0,C 0,E1 0.1598,E2 90.0717} C_DIS
LIN {X 6.9015,Y -4.9387,Z 34,A -2.662,B 0,C 0,E1 0.1598,E2 90.0717} C_DIS
LIN {X 7.356,Y -4.2325,Z 34,A -2.6151,B 0,C 0,E1 0.1598,E2 90.0718} C_DIS
LIN {X 7.7386,Y -3.4849,Z 34,A -2.5692,B 0,C 0,E1 0.1598,E2 90.0718} C_DIS
LIN {X 8.0454,Y -2.7031,Z 34,A -2.5245,B 0,C 0,E1 0.1598,E2 90.0718} C_DIS
LIN {X 8.3206,Y -1.6901,Z 34,A -2.4709,B 0,C 0,E1 0.1598,E2 90.0716} C_DIS
LIN {X 8.4678,Y -0.5877,Z 34,A -2.4184,B 0,C 0,E1 0.1598,E2 90.0716} C_DIS
LIN {X 8.4723,Y 0.5556,Z 34,A -2.3694,B 0,C 0,E1 0.1598,E2 90.0716} C_DIS
LIN {X 8.3305,Y 1.6275,Z 34,A -2.3291,B 0,C 0,E1 0.1598,E2 90.0718} C_DIS
LIN {X 8.1219,Y 2.4671,Z 34,A -2.3012,B 0,C 0,E1 0.1598,E2 90.0721} C_DIS
LIN {X 7.8287,Y 3.2809,Z 34,A -2.2773,B 0,C 0,E1 0.1598,E2 90.0721} C_DIS
LIN {X 7.454,Y 4.0606,Z 34,A -2.258,B 0,C 0,E1 0.1598,E2 90.0721} C_DIS
LIN {X 7.0018,Y 4.7981,Z 34,A -2.2433,B 0,C 0,E1 0.1598,E2 90.0722} C_DIS
LIN {X 6.4771,Y 5.4858,Z 34,A -2.2334,B 0,C 0,E1 0.1598,E2 90.0723} C_DIS
LIN {X 5.8853,Y 6.1168,Z 34,A -2.2284,B 0,C 0,E1 0.1598,E2 90.0723} C_DIS
LIN {X 4.904,Y 6.9311,Z 34,A -2.2299,B 0,C 0,E1 0.1598,E2 90.0723} C_DIS
LIN {X 3.8701,Y 7.5537,Z 34,A -2.2417,B 0,C 0,E1 0.1598,E2 90.0723} C_DIS
LIN {X 3.0887,Y 7.9055,Z 34,A -2.2558,B 0,C 0,E1 0.1598,E2 90.0725} C_DIS
LIN {X 2.2759,Y 8.1768,Z 34,A -2.2744,B 0,C 0,E1 0.1598,E2 90.0725} C_DIS
LIN {X 1.4399,Y 8.3652,Z 34,A -2.2973,B 0,C 0,E1 0.1598,E2 90.0725} C_DIS
LIN {X 0.3754,Y 8.4839,Z 34,A -2.3316,B 0,C 0,E1 0.1598,E2 90.0725} C_DIS
LIN {X -0.8692,Y 8.4434,Z 34,A -2.3793,B 0,C 0,E1 0.1598,E2 90.0724} C_DIS
LIN {X -1.6355,Y 8.3321,Z 34,A -2.4123,B 0,C 0,E1 0.1598,E2 90.0724} C_DIS
LIN {X -2.9404,Y 7.9648,Z 34,A -2.4759,B 0,C 0,E1 0.1598,E2 90.0722} C_DIS
LIN {X -4.0526,Y 7.458,Z 34,A -2.5383,B 0,C 0,E1 0.1598,E2 90.0721} C_DIS
LIN {X -4.8087,Y 6.9935,Z 34,A -2.5859,B 0,C 0,E1 0.1598,E2 90.0721} C_DIS
LIN {X -5.5123,Y 6.4527,Z 34,A -2.6346,B 0,C 0,E1 0.1598,E2 90.0719} C_DIS
LIN {X -6.1559,Y 5.8419,Z 34,A -2.6841,B 0,C 0,E1 0.1598,E2 90.0719} C_DIS
LIN {X -6.8695,Y 4.9926,Z 34,A -2.7461,B 0,C 0,E1 0.1598,E2 90.0715} C_DIS
LIN {X -7.5089,Y 3.9553,Z 34,A -2.8132,B 0,C 0,E1 0.1598,E2 90.0712} C_DIS
LIN {X -7.8787,Y 3.1535,Z 34,A -2.861,B 0,C 0,E1 0.1598,E2 90.0714} C_DIS
LIN {X -8.2251,Y 2.1057,Z 34,A -2.9176,B 0,C 0,E1 0.1598,E2 90.071} C_DIS
LIN {X -8.4385,Y 0.9201,Z 34,A -2.9754,B 0,C 0,E1 0.1598,E2 90.0708} C_DIS
LIN {X -8.4884,Y 0.1937,Z 34,A -3.0083,B 0,C 0,E1 0.1598,E2 90.0712} C_DIS
LIN {X -8.4473,Y -0.8601,Z 34,A -3.0511,B 0,C 0,E1 0.1598,E2 90.0709} C_DIS
LIN {X -8.266,Y -1.9185,Z 34,A -3.0892,B 0,C 0,E1 0.1598,E2 90.0709} C_DIS
LIN {X -8.0303,Y -2.7443,Z 34,A -3.1156,B 0,C 0,E1 0.1598,E2 90.0711} C_DIS
LIN {X -7.712,Y -3.5421,Z 34,A -3.1377,B 0,C 0,E1 0.1598,E2 90.0711} C_DIS
LIN {X -7.3144,Y -4.3034,Z 34,A -3.1553,B 0,C 0,E1 0.1598,E2 90.0711} C_DIS
LIN {X -6.8418,Y -5.0206,Z 34,A -3.1683,B 0,C 0,E1 0.1598,E2 90.0711} C_DIS
LIN {X -6.2991,Y -5.6864,Z 34,A -3.1766,B 0,C 0,E1 0.1598,E2 90.0711} C_DIS
LIN {X -5.6919,Y -6.2939,Z 34,A -3.1801,B 0,C 0,E1 0.1598,E2 90.0711} C_DIS
LIN {X -5.0265,Y -6.837,Z 34,A -3.1788,B 0,C 0,E1 0.1598,E2 90.0711} C_DIS
LIN {X -4.3097,Y -7.3102,Z 34,A -3.1726,B 0,C 0,E1 0.1598,E2 90.0712} C_DIS
LIN {X -3.5487,Y -7.7086,Z 34,A -3.1616,B 0,C 0,E1 0.1598,E2 90.0712} C_DIS
LIN {X -2.7514,Y -8.0281,Z 34,A -3.146,B 0,C 0,E1 0.1598,E2 90.0713} C_DIS
LIN {X -1.9258,Y -8.2655,Z 34,A -3.1258,B 0,C 0,E1 0.1598,E2 90.0713} C_DIS
LIN {X -1.0806,Y -8.4186,Z 34,A -3.1014,B 0,C 0,E1 0.1598,E2 90.0714} C_DIS
LIN {X -0.0093,Y -8.4875,Z 34,A -3.0651,B 0,C 0,E1 0.1598,E2 90.0714} C_DIS
Enddeposition()
LIN {X 0.0007,Y -4.7533,Z 35,A -2.8912,B 0,C 0,E1 0.1598,E2 90.0604} C_DIS
Startdeposition()
$VEL.CP = VEL_PRINT
LIN {X 0.0007,Y -4.7533,Z 35,A -2.8969,B 0,C 0,E1 0.1598,E2 90.0661} C_DIS
LIN {X -0.8335,Y -4.6781,Z 35,A -2.9292,B 0,C 0,E1 0.1598,E2 90.071} C_DIS
LIN {X -1.4836,Y -4.5146,Z 35,A -2.9467,B 0,C 0,E1 0.1598,E2 90.0716} C_DIS
LIN {X -2.1044,Y -4.2616,Z 35,A -2.9588,B 0,C 0,E1 0.1598,E2 90.0716} C_DIS
LIN {X -2.6829,Y -3.9227,Z 35,A -2.9656,B 0,C 0,E1 0.1598,E2 90.0716} C_DIS
LIN {X -3.208,Y -3.5058,Z 35,A -2.9672,B 0,C 0,E1 0.1598,E2 90.0716} C_DIS
LIN {X -3.6685,Y -3.0186,Z 35,A -2.9634,B 0,C 0,E1 0.1598,E2 90.0715} C_DIS
LIN {X -4.0568,Y -2.4723,Z 35,A -2.9545,B 0,C 0,E1 0.1598,E2 90.0715} C_DIS
LIN {X -4.3656,Y -1.8773,Z 35,A -2.9406,B 0,C 0,E1 0.1598,E2 90.0715} C_DIS
LIN {X -4.5845,Y -1.2437,Z 35,A -2.9218,B 0,C 0,E1 0.1598,E2 90.0715} C_DIS
LIN {X -4.7139,Y -0.5861,Z 35,A -2.8987,B 0,C 0,E1 0.1598,E2 90.0715} C_DIS
LIN {X -4.7498,Y 0.0831,Z 35,A -2.8717,B 0,C 0,E1 0.1598,E2 90.0715} C_DIS
LIN {X -4.6913,Y 0.7507,Z 35,A -2.8413,B 0,C 0,E1 0.1598,E2 90.0715} C_DIS
LIN {X -4.5378,Y 1.4031,Z 35,A -2.808,B 0,C 0,E1 0.1598,E2 90.0716} C_DIS
LIN {X -4.2964,Y 2.0282,Z 35,A -2.7727,B 0,C 0,E1 0.1598,E2 90.0716} C_DIS
LIN {X -3.9692,Y 2.6134,Z 35,A -2.7359,B 0,C 0,E1 0.1598,E2 90.0717} C_DIS
LIN {X -3.5609,Y 3.1451,Z 35,A -2.6984,B 0,C 0,E1 0.1598,E2 90.0718} C_DIS
LIN {X -3.0837,Y 3.6158,Z 35,A -2.6609,B 0,C 0,E1 0.1598,E2 90.0719} C_DIS
LIN {X -2.5441,Y 4.0139,Z 35,A -2.6242,B 0,C 0,E1 0.1598,E2 90.0719} C_DIS
LIN {X -1.9537,Y 4.3312,Z 35,A -2.5891,B 0,C 0,E1 0.1598,E2 90.0721} C_DIS
LIN {X -1.3248,Y 4.5637,Z 35,A -2.5561,B 0,C 0,E1 0.1598,E2 90.0721} C_DIS
LIN {X -0.6691,Y 4.7025,Z 35,A -2.526,B 0,C 0,E1 0.1598,E2 90.0721} C_DIS
LIN {X -0.0007,Y 4.7512,Z 35,A -2.4993,B 0,C 0,E1 0.1598,E2 90.0722} C_DIS
LIN {X 0.6678,Y 4.7037,Z 35,A -2.4767,B 0,C 0,E1 0.1598,E2 90.0722} C_DIS
LIN {X 1.323,Y 4.5627,Z 35,A -2.4585,B 0,C 0,E1 0.1598,E2 90.0722} C_DIS
LIN {X 1.952,Y 4.3314,Z 35,A -2.4451,B 0,C 0,E1 0.1598,E2 90.0722} C_DIS
LIN {X 2.542,Y 4.0132,Z 35,A -2.4369,B 0,C 0,E1 0.1598,E2 90.0722} C_DIS
LIN {X 3.0811,Y 3.6151,Z 35,A -2.4339,B 0,C 0,E1 0.1598,E2 90.0722} C_DIS
LIN {X 3.5597,Y 3.146,Z 35,A -2.4361,B 0,C 0,E1 0.1598,E2 90.0722} C_DIS
LIN {X 3.9673,Y 2.6138,Z 35,A -2.4437,B 0,C 0,E1 0.1598,E2 90.0722} C_DIS
LIN {X 4.2968,Y 2.0301,Z 35,A -2.4564,B 0,C 0,E1 0.1598,E2 90.0721} C_DIS
LIN {X 4.5402,Y 1.4054,Z 35,A -2.4739,B 0,C 0,E1 0.1598,E2 90.0721} C_DIS
LIN {X 4.6927,Y 0.7526,Z 35,A -2.4961,B 0,C 0,E1 0.1598,E2 90.072} C_DIS
LIN {X 4.7518,Y 0.0847,Z 35,A -2.5223,B 0,C 0,E1 0.1598,E2 90.072} C_DIS
LIN {X 4.7028,Y -0.6675,Z 35,A -2.556,B 0,C 0,E1 0.1598,E2 90.0718} C_DIS
LIN {X 4.5852,Y -1.2421,Z 35,A -2.585,B 0,C 0,E1 0.1598,E2 90.072} C_DIS
LIN {X 4.366,Y -1.8755,Z 35,A -2.6199,B 0,C 0,E1 0.1598,E2 90.0719} C_DIS
LIN {X 4.0574,Y -2.4705,Z 35,A -2.6566,B 0,C 0,E1 0.1598,E2 90.0719} C_DIS
LIN {X 3.6688,Y -3.0164,Z 35,A -2.6942,B 0,C 0,E1 0.1598,E2 90.0719} C_DIS
LIN {X 3.2093,Y -3.5044,Z 35,A -2.7319,B 0,C 0,E1 0.1598,E2 90.0719} C_DIS
LIN {X 2.6832,Y -3.9199,Z 35,A -2.7689,B 0,C 0,E1 0.1598,E2 90.0718} C_DIS
LIN {X 2.1046,Y -4.2582,Z 35,A -2.8045,B 0,C 0,E1 0.1598,E2 90.0718} C_DIS
LIN {X 1.4846,Y -4.5125,Z 35,A -2.8382,B 0,C 0,E1 0.1598,E2 90.0718} C_DIS
LIN {X 0.8348,Y -4.6768,Z 35,A -2.869,B 0,C 0,E1 0.1598,E2 90.0718} C_DIS
LIN {X 0.0007,Y -4.7533,Z 35,A -2.9029,B 0,C 0,E1 0.1598,E2 90.0718} C_DIS
Enddeposition()
LIN {X 0.0007,Y -4.7533,Z 35,A -2.9029,B 0,C 0,E1 0.1598,E2 90.0718} C_DIS
Startdeposition()
$VEL.CP = VEL_PRINT
LIN {X 0.6321,Y -5.6506,Z 35,A -2.9174,B 0,C 0,E1 0.1598,E2 90.0711} C_DIS
LIN {X 1.416,Y -5.5056,Z 35,A -2.883,B 0,C 0,E1 0.1598,E2 90.0717} C_DIS
LIN {X 2.1724,Y -5.2538,Z 35,A -2.8445,B 0,C 0,E1 0.1598,E2 90.0717} C_DIS
LIN {X 2.8848,Y -4.8961,Z 35,A -2.8031,B 0,C 0,E1 0.1598,E2 90.0717} C_DIS
LIN {X 3.5408,Y -4.4438,Z 35,A -2.7598,B 0,C 0,E1 0.1598,E2 90.0717} C_DIS
LIN {X 4.1277,Y -3.9049,Z 35,A -2.7152,B 0,C 0,E1 0.1598,E2 90.0718} C_DIS
LIN {X 4.6349,Y -3.2903,Z 35,A -2.6704,B 0,C 0,E1 0.1598,E2 90.0718} C_DIS
LIN {X 5.0495,Y -2.6095,Z 35,A -2.6261,B 0,C 0,E1 0.1598,E2 90.0718} C_DIS
LIN {X 5.3636,Y -1.8772,Z 35,A -2.5833,B 0,C 0,E1 0.1598,E2 90.0718} C_DIS
LIN {X 5.5731,Y -1.1085,Z 35,A -2.5429,B 0,C 0,E1 0.1598,E2 90.0718} C_DIS
LIN {X 5.6906,Y 0.0256,Z 35,A -2.4899,B 0,C 0,E1 0.1598,E2 90.0716} C_DIS
LIN {X 5.5568,Y 1.2229,Z 35,A -2.4436,B 0,C 0,E1 0.1598,E2 90.0714} C_DIS
LIN {X 5.196,Y 2.3041,Z 35,A -2.4111,B 0,C 0,E1 0.1598,E2 90.0716} C_DIS
LIN {X 4.801,Y 3.0392,Z 35,A -2.3947,B 0,C 0,E1 0.1598,E2 90.072} C_DIS
LIN {X 4.3042,Y 3.7097,Z 35,A -2.3846,B 0,C 0,E1 0.1598,E2 90.0721} C_DIS
LIN {X 3.7145,Y 4.3,Z 35,A -2.3813,B 0,C 0,E1 0.1598,E2 90.0721} C_DIS
LIN {X 3.0442,Y 4.7971,Z 35,A -2.3849,B 0,C 0,E1 0.1598,E2 90.0722} C_DIS
LIN {X 2.3089,Y 5.1915,Z 35,A -2.3954,B 0,C 0,E1 0.1598,E2 90.0722} C_DIS
LIN {X 1.5236,Y 5.4737,Z 35,A -2.4124,B 0,C 0,E1 0.1598,E2 90.0722} C_DIS
LIN {X 0.7058,Y 5.6389,Z 35,A -2.4356,B 0,C 0,E1 0.1598,E2 90.0723} C_DIS
LIN {X -0.1278,Y 5.6826,Z 35,A -2.4645,B 0,C 0,E1 0.1598,E2 90.0723} C_DIS
LIN {X -0.9589,Y 5.6042,Z 35,A -2.4984,B 0,C 0,E1 0.1598,E2 90.0723} C_DIS
LIN {X -1.7692,Y 5.4032,Z 35,A -2.5368,B 0,C 0,E1 0.1598,E2 90.0722} C_DIS
LIN {X -2.5403,Y 5.0837,Z 35,A -2.5788,B 0,C 0,E1 0.1598,E2 90.0721} C_DIS
LIN {X -3.2576,Y 4.657,Z 35,A -2.6232,B 0,C 0,E1 0.1598,E2 90.072} C_DIS
LIN {X -3.9044,Y 4.1296,Z 35,A -2.6693,B 0,C 0,E1 0.1598,E2 90.0719} C_DIS
LIN {X -4.4681,Y 3.514,Z 35,A -2.7161,B 0,C 0,E1 0.1598,E2 90.0718} C_DIS
LIN {X -4.9348,Y 2.8218,Z 35,A -2.7625,B 0,C 0,E1 0.1598,E2 90.0716} C_DIS
LIN {X -5.2935,Y 2.0682,Z 35,A -2.8075,B 0,C 0,E1 0.1598,E2 90.0716} C_DIS
LIN {X -5.5416,Y 1.2711,Z 35,A -2.8503,B 0,C 0,E1 0.1598,E2 90.0714} C_DIS
LIN {X -5.6673,Y 0.4457,Z 35,A -2.8898,B 0,C 0,E1 0.1598,E2 90.0714} C_DIS
LIN {X -5.6704,Y -0.389,Z 35,A -2.9252,B 0,C 0,E1 0.1598,E2 90.0714} C_DIS
LIN {X -5.5519,Y -1.2152,Z 35,A -2.9558,B 0,C 0,E1 0.1598,E2 90.0713} C_DIS
LIN {X -5.3139,Y -2.0151,Z 35,A -2.981,B 0,C 0,E1 0.1598,E2 90.0713} C_DIS
LIN {X -4.9625,Y -2.7722,Z 35,A -3.0001,B 0,C 0,E1 0.1598,E2 90.0713} C_DIS
LIN {X -4.503,Y -3.469,Z 35,A -3.0128,B 0,C 0,E1 0.1598,E2 90.0713} C_DIS
LIN {X -3.9476,Y -4.0924,Z 35,A -3.0189,B 0,C 0,E1 0.1598,E2 90.0713} C_DIS
LIN {X -3.1359,Y -4.7484,Z 35,A -3.0169,B 0,C 0,E1 0.1598,E2 90.0713} C_DIS
LIN {X -2.2606,Y -5.2208,Z 35,A -3.0049,B 0,C 0,E1 0.1598,E2 90.0714} C_DIS
LIN {X -0.9938,Y -5.6028,Z 35,A -2.9747,B 0,C 0,E1 0.1598,E2 90.0715} C_DIS
LIN {X -0.3523,Y -5.6754,Z 35,A -2.9543,B 0,C 0,E1 0.1598,E2 90.0716} C_DIS
LIN {X -0.3523,Y -5.6754,Z 35,A -2.9543,B 0,C 0,E1 0.1598,E2 90.0716} C_DIS
Enddeposition()
LIN {X 0.0424,Y -6.6204,Z 35,A -2.979,B 0,C 0,E1 0.1598,E2 90.0704} C_DIS
Startdeposition()
$VEL.CP = VEL_PRINT
LIN {X -0.8658,Y -6.563,Z 35,A -3.011,B 0,C 0,E1 0.1598,E2 90.0715} C_DIS
LIN {X -1.5812,Y -6.4272,Z 35,A -3.0315,B 0,C 0,E1 0.1598,E2 90.0715} C_DIS
LIN {X -2.2782,Y -6.216,Z 35,A -3.0481,B 0,C 0,E1 0.1598,E2 90.0715} C_DIS
LIN {X -2.9475,Y -5.929,Z 35,A -3.0604,B 0,C 0,E1 0.1598,E2 90.0715} C_DIS
LIN {X -3.5804,Y -5.5689,Z 35,A -3.0683,B 0,C 0,E1 0.1598,E2 90.0715} C_DIS
LIN {X -4.1691,Y -5.1405,Z 35,A -3.0717,B 0,C 0,E1 0.1598,E2 90.0714} C_DIS
LIN {X -4.7092,Y -4.6519,Z 35,A -3.0708,B 0,C 0,E1 0.1598,E2 90.0714} C_DIS
LIN {X -5.1917,Y -4.1064,Z 35,A -3.0654,B 0,C 0,E1 0.1598,E2 90.0714} C_DIS
LIN {X -5.6121,Y -3.5116,Z 35,A -3.0556,B 0,C 0,E1 0.1598,E2 90.0714} C_DIS
LIN {X -5.9651,Y -2.8748,Z 35,A -3.0416,B 0,C 0,E1 0.1598,E2 90.0713} C_DIS
LIN {X -6.2428,Y -2.2015,Z 35,A -3.0233,B 0,C 0,E1 0.1598,E2 90.0713} C_DIS
LIN {X -6.4457,Y -1.5023,Z 35,A -3.0011,B 0,C 0,E1 0.1598,E2 90.0713} C_DIS
LIN {X -6.5737,Y -0.7853,Z 35,A -2.9755,B 0,C 0,E1 0.1598,E2 90.0713} C_DIS
LIN {X -6.6202,Y -0.0587,Z 35,A -2.9465,B 0,C 0,E1 0.1598,E2 90.0713} C_DIS
LIN {X -6.5497,Y 0.9862,Z 35,A -2.8994,B 0,C 0,E1 0.1598,E2 90.0712} C_DIS
LIN {X -6.3398,Y 1.8992,Z 35,A -2.8532,B 0,C 0,E1 0.1598,E2 90.0714} C_DIS
LIN {X -6.0842,Y 2.6035,Z 35,A -2.8142,B 0,C 0,E1 0.1598,E2 90.0716} C_DIS
LIN {X -5.7515,Y 3.2749,Z 35,A -2.7736,B 0,C 0,E1 0.1598,E2 90.0716} C_DIS
LIN {X -5.3445,Y 3.9041,Z 35,A -2.732,B 0,C 0,E1 0.1598,E2 90.0717} C_DIS
LIN {X -4.87,Y 4.484,Z 35,A -2.69,B 0,C 0,E1 0.1598,E2 90.0718} C_DIS
LIN {X -4.3311,Y 5.0048,Z 35,A -2.6482,B 0,C 0,E1 0.1598,E2 90.0719} C_DIS
LIN {X -3.7372,Y 5.4616,Z 35,A -2.607,B 0,C 0,E1 0.1598,E2 90.0719} C_DIS
LIN {X -3.0967,Y 5.8507,Z 35,A -2.5669,B 0,C 0,E1 0.1598,E2 90.0721} C_DIS
LIN {X -2.4157,Y 6.1638,Z 35,A -2.5286,B 0,C 0,E1 0.1598,E2 90.0721} C_DIS
LIN {X -1.7032,Y 6.3963,Z 35,A -2.4925,B 0,C 0,E1 0.1598,E2 90.0722} C_DIS
LIN {X -0.9692,Y 6.5473,Z 35,A -2.459,B 0,C 0,E1 0.1598,E2 90.0722} C_DIS
LIN {X -0.223,Y 6.6156,Z 35,A -2.4286,B 0,C 0,E1 0.1598,E2 90.0723} C_DIS
LIN {X 0.5261,Y 6.5979,Z 35,A -2.4017,B 0,C 0,E1 0.1598,E2 90.0723} C_DIS
LIN {X 1.2685,Y 6.4964,Z 35,A -2.3786,B 0,C 0,E1 0.1598,E2 90.0723} C_DIS
LIN {X 1.995,Y 6.3125,Z 35,A -2.3596,B 0,C 0,E1 0.1598,E2 90.0723} C_DIS
LIN {X 2.6955,Y 6.046,Z 35,A -2.3451,B 0,C 0,E1 0.1598,E2 90.0723} C_DIS
LIN {X 3.3617,Y 5.7027,Z 35,A -2.335,B 0,C 0,E1 0.1598,E2 90.0723} C_DIS
LIN {X 4.2408,Y 5.0876,Z 35,A -2.3286,B 0,C 0,E1 0.1598,E2 90.0723} C_DIS
LIN {X 4.9002,Y 4.4497,Z 35,A -2.3314,B 0,C 0,E1 0.1598,E2 90.0723} C_DIS
LIN {X 5.3628,Y 3.8799,Z 35,A -2.3386,B 0,C 0,E1 0.1598,E2 90.0723} C_DIS
LIN {X 5.7596,Y 3.2627,Z 35,A -2.3502,B 0,C 0,E1 0.1598,E2 90.0723} C_DIS
LIN {X 6.0876,Y 2.606,Z 35,A -2.366,B 0,C 0,E1 0.1598,E2 90.0722} C_DIS
LIN {X 6.3353,Y 1.9151,Z 35,A -2.3863,B 0,C 0,E1 0.1598,E2 90.0722} C_DIS
LIN {X 6.5092,Y 1.2021,Z 35,A -2.4102,B 0,C 0,E1 0.1598,E2 90.0721} C_DIS
LIN {X 6.6012,Y 0.4741,Z 35,A -2.4379,B 0,C 0,E1 0.1598,E2 90.0721} C_DIS
LIN {X 6.6141,Y -0.2596,Z 35,A -2.4686,B 0,C 0,E1 0.1598,E2 90.072} C_DIS
LIN {X 6.544,Y -0.99,Z 35,A -2.5023,B 0,C 0,E1 0.1598,E2 90.072} C_DIS
LIN {X 6.3958,Y -1.7088,Z 35,A -2.5384,B 0,C 0,E1 0.1598,E2 90.072} C_DIS
LIN {X 6.1661,Y -2.4059,Z 35,A -2.5766,B 0,C 0,E1 0.1598,E2 90.0719} C_DIS
LIN {X 5.863,Y -3.0743,Z 35,A -2.6162,B 0,C 0,E1 0.1598,E2 90.0719} C_DIS
LIN {X 5.4858,Y -3.704,Z 35,A -2.6569,B 0,C 0,E1 0.1598,E2 90.0719} C_DIS
LIN {X 5.044,Y -4.2902,Z 35,A -2.6981,B 0,C 0,E1 0.1598,E2 90.0718} C_DIS
LIN {X 4.5382,Y -4.8221,Z 35,A -2.7394,B 0,C 0,E1 0.1598,E2 90.0718} C_DIS
LIN {X 3.9762,Y -5.294,Z 35,A -2.7802,B 0,C 0,E1 0.1598,E2 90.0718} C_DIS
LIN {X 3.3646,Y -5.6999,Z 35,A -2.8199,B 0,C 0,E1 0.1598,E2 90.0718} C_DIS
LIN {X 2.7132,Y -6.0379,Z 35,A -2.8582,B 0,C 0,E1 0.1598,E2 90.0718} C_DIS
LIN {X 2.0289,Y -6.3029,Z 35,A -2.8946,B 0,C 0,E1 0.1598,E2 90.0717} C_DIS
LIN {X 1.3187,Y -6.4881,Z 35,A -2.9286,B 0,C 0,E1 0.1598,E2 90.0717} C_DIS
LIN {X 0.5922,Y -6.5927,Z 35,A -2.9597,B 0,C 0,E1 0.1598,E2 90.0717} C_DIS
LIN {X 0.5922,Y -6.5927,Z 35,A -2.9597,B 0,C 0,E1 0.1598,E2 90.0717} C_DIS
Enddeposition()
LIN {X 0.0388,Y -7.5538,Z 35,A -3.0198,B 0,C 0,E1 0.1598,E2 90.0704} C_DIS
Startdeposition()
$VEL.CP = VEL_PRINT
LIN {X 0.7843,Y -7.5163,Z 35,A -2.992,B 0,C 0,E1 0.1598,E2 90.0715} C_DIS
LIN {X 1.871,Y -7.318,Z 35,A -2.9438,B 0,C 0,E1 0.1598,E2 90.0716} C_DIS
LIN {X 2.713,Y -7.0494,Z 35,A -2.9015,B 0,C 0,E1 0.1598,E2 90.0716} C_DIS
LIN {X 3.7739,Y -6.5479,Z 35,A -2.8411,B 0,C 0,E1 0.1598,E2 90.0716} C_DIS
LIN {X 4.8287,Y -5.8074,Z 35,A -2.7707,B 0,C 0,E1 0.1598,E2 90.0716} C_DIS
LIN {X 5.674,Y -4.9916,Z 35,A -2.7049,B 0,C 0,E1 0.1598,E2 90.0716} C_DIS
LIN {X 6.2216,Y -4.284,Z 35,A -2.6547,B 0,C 0,E1 0.1598,E2 90.0718} C_DIS
LIN {X 6.6001,Y -3.6765,Z 35,A -2.6149,B 0,C 0,E1 0.1598,E2 90.0718} C_DIS
LIN {X 6.9904,Y -2.8713,Z 35,A -2.5661,B 0,C 0,E1 0.1598,E2 90.0718} C_DIS
LIN {X 7.3101,Y -1.9147,Z 35,A -2.5135,B 0,C 0,E1 0.1598,E2 90.0718} C_DIS
LIN {X 7.5037,Y -0.8955,Z 35,A -2.4628,B 0,C 0,E1 0.1598,E2 90.0718} C_DIS
LIN {X 7.5586,Y 0.0013,Z 35,A -2.4227,B 0,C 0,E1 0.1598,E2 90.0719} C_DIS
LIN {X 7.4921,Y 0.9979,Z 35,A -2.3825,B 0,C 0,E1 0.1598,E2 90.0719} C_DIS
LIN {X 7.2568,Y 2.1127,Z 35,A -2.3435,B 0,C 0,E1 0.1598,E2 90.0717} C_DIS
LIN {X 6.8549,Y 3.1826,Z 35,A -2.3128,B 0,C 0,E1 0.1598,E2 90.0718} C_DIS
LIN {X 6.4122,Y 3.993,Z 35,A -2.2949,B 0,C 0,E1 0.1598,E2 90.0721} C_DIS
LIN {X 5.7868,Y 4.8598,Z 35,A -2.281,B 0,C 0,E1 0.1598,E2 90.0721} C_DIS
LIN {X 5.151,Y 5.5233,Z 35,A -2.2764,B 0,C 0,E1 0.1598,E2 90.0723} C_DIS
LIN {X 4.5888,Y 5.9972,Z 35,A -2.2771,B 0,C 0,E1 0.1598,E2 90.0723} C_DIS
LIN {X 3.8301,Y 6.516,Z 35,A -2.283,B 0,C 0,E1 0.1598,E2 90.0723} C_DIS
LIN {X 2.7967,Y 7.022,Z 35,A -2.2997,B 0,C 0,E1 0.1598,E2 90.0723} C_DIS
LIN {X 1.1634,Y 7.4668,Z 35,A -2.3412,B 0,C 0,E1 0.1598,E2 90.0723} C_DIS
LIN {X -0.5224,Y 7.5388,Z 35,A -2.4004,B 0,C 0,E1 0.1598,E2 90.0723} C_DIS
LIN {X -1.671,Y 7.3707,Z 35,A -2.45,B 0,C 0,E1 0.1598,E2 90.0723} C_DIS
LIN {X -2.8313,Y 7.0027,Z 35,A -2.5083,B 0,C 0,E1 0.1598,E2 90.0722} C_DIS
LIN {X -3.6424,Y 6.6207,Z 35,A -2.5543,B 0,C 0,E1 0.1598,E2 90.0721} C_DIS
LIN {X -4.5769,Y 6.0128,Z 35,A -2.6144,B 0,C 0,E1 0.1598,E2 90.0719} C_DIS
LIN {X -5.468,Y 5.2154,Z 35,A -2.6809,B 0,C 0,E1 0.1598,E2 90.0717} C_DIS
LIN {X -6.2551,Y 4.24,Z 35,A -2.7509,B 0,C 0,E1 0.1598,E2 90.0714} C_DIS
LIN {X -6.7964,Y 3.2937,Z 35,A -2.8108,B 0,C 0,E1 0.1598,E2 90.0714} C_DIS
LIN {X -7.2172,Y 2.2396,Z 35,A -2.8707,B 0,C 0,E1 0.1598,E2 90.0712} C_DIS
LIN {X -7.4753,Y 1.0884,Z 35,A -2.9287,B 0,C 0,E1 0.1598,E2 90.0709} C_DIS
LIN {X -7.5501,Y 0.3549,Z 35,A -2.9628,B 0,C 0,E1 0.1598,E2 90.0712} C_DIS
LIN {X -7.4927,Y -0.9923,Z 35,A -3.0172,B 0,C 0,E1 0.1598,E2 90.0707} C_DIS
LIN {X -7.3118,Y -1.8997,Z 35,A -3.0493,B 0,C 0,E1 0.1598,E2 90.0711} C_DIS
LIN {X -7.0908,Y -2.6062,Z 35,A -3.0712,B 0,C 0,E1 0.1598,E2 90.0712} C_DIS
LIN {X -6.8014,Y -3.2875,Z 35,A -3.0894,B 0,C 0,E1 0.1598,E2 90.0712} C_DIS
LIN {X -6.4471,Y -3.9374,Z 35,A -3.1039,B 0,C 0,E1 0.1598,E2 90.0712} C_DIS
LIN {X -6.0295,Y -4.5486,Z 35,A -3.1145,B 0,C 0,E1 0.1598,E2 90.0712} C_DIS
LIN {X -5.4311,Y -5.2542,Z 35,A -3.1223,B 0,C 0,E1 0.1598,E2 90.0712} C_DIS
LIN {X -4.6325,Y -5.9668,Z 35,A -3.1232,B 0,C 0,E1 0.1598,E2 90.0712} C_DIS
LIN {X -4.0165,Y -6.3944,Z 35,A -3.119,B 0,C 0,E1 0.1598,E2 90.0713} C_DIS
LIN {X -3.364,Y -6.764,Z 35,A -3.1107,B 0,C 0,E1 0.1598,E2 90.0713} C_DIS
LIN {X -2.677,Y -7.0648,Z 35,A -3.0983,B 0,C 0,E1 0.1598,E2 90.0713} C_DIS
LIN {X -1.7822,Y -7.3446,Z 35,A -3.0774,B 0,C 0,E1 0.1598,E2 90.0714} C_DIS
LIN {X -0.7664,Y -7.5184,Z 35,A -3.0476,B 0,C 0,E1 0.1598,E2 90.0714} C_DIS
LIN {X 0.0388,Y -7.5538,Z 35,A -3.0196,B 0,C 0,E1 0.1598,E2 90.0715} C_DIS
Enddeposition()
LIN {X 0.0388,Y -7.5538,Z 35,A -3.0196,B 0,C 0,E1 0.1598,E2 90.0715} C_DIS
Startdeposition()
$VEL.CP = VEL_PRINT
LIN {X -0.6219,Y -8.4655,Z 35,A -3.0822,B 0,C 0,E1 0.1598,E2 90.0709} C_DIS
LIN {X -1.4764,Y -8.3584,Z 35,A -3.1095,B 0,C 0,E1 0.1598,E2 90.0714} C_DIS
LIN {X -2.3158,Y -8.1653,Z 35,A -3.1321,B 0,C 0,E1 0.1598,E2 90.0714} C_DIS
LIN {X -3.1312,Y -7.8881,Z 35,A -3.1502,B 0,C 0,E1 0.1598,E2 90.0714} C_DIS
LIN {X -3.9144,Y -7.5299,Z 35,A -3.1636,B 0,C 0,E1 0.1598,E2 90.0713} C_DIS
LIN {X -4.6572,Y -7.0942,Z 35,A -3.1724,B 0,C 0,E1 0.1598,E2 90.0713} C_DIS
LIN {X -5.3522,Y -6.5856,Z 35,A -3.1762,B 0,C 0,E1 0.1598,E2 90.0712} C_DIS
LIN {X -5.992,Y -6.0092,Z 35,A -3.1752,B 0,C 0,E1 0.1598,E2 90.0712} C_DIS
LIN {X -6.5703,Y -5.3712,Z 35,A -3.1694,B 0,C 0,E1 0.1598,E2 90.0712} C_DIS
LIN {X -7.0809,Y -4.6778,Z 35,A -3.1587,B 0,C 0,E1 0.1598,E2 90.0712} C_DIS
LIN {X -7.5186,Y -3.9362,Z 35,A -3.1434,B 0,C 0,E1 0.1598,E2 90.0711} C_DIS
LIN {X -7.8787,Y -3.1539,Z 35,A -3.1235,B 0,C 0,E1 0.1598,E2 90.0711} C_DIS
LIN {X -8.1574,Y -2.3392,Z 35,A -3.0993,B 0,C 0,E1 0.1598,E2 90.0711} C_DIS
LIN {X -8.3522,Y -1.5004,Z 35,A -3.0709,B 0,C 0,E1 0.1598,E2 90.0711} C_DIS
LIN {X -8.4864,Y -0.2829,Z 35,A -3.0241,B 0,C 0,E1 0.1598,E2 90.0708} C_DIS
LIN {X -8.4402,Y 0.896,Z 35,A -2.9726,B 0,C 0,E1 0.1598,E2 90.0709} C_DIS
LIN {X -8.2248,Y 2.1069,Z 35,A -2.9135,B 0,C 0,E1 0.1598,E2 90.0709} C_DIS
LIN {X -7.8778,Y 3.1556,Z 35,A -2.8566,B 0,C 0,E1 0.1598,E2 90.0712} C_DIS
LIN {X -7.5074,Y 3.958,Z 35,A -2.8093,B 0,C 0,E1 0.1598,E2 90.0715} C_DIS
LIN {X -6.8725,Y 4.9885,Z 35,A -2.7422,B 0,C 0,E1 0.1598,E2 90.0715} C_DIS
LIN {X -6.1228,Y 5.878,Z 35,A -2.6771,B 0,C 0,E1 0.1598,E2 90.0715} C_DIS
LIN {X -5.4841,Y 6.4775,Z 35,A -2.6284,B 0,C 0,E1 0.1598,E2 90.0719} C_DIS
LIN {X -4.7876,Y 7.0085,Z 35,A -2.5803,B 0,C 0,E1 0.1598,E2 90.0719} C_DIS
LIN {X -4.04,Y 7.4651,Z 35,A -2.5335,B 0,C 0,E1 0.1598,E2 90.0721} C_DIS
LIN {X -2.9421,Y 7.9641,Z 35,A -2.4719,B 0,C 0,E1 0.1598,E2 90.0721} C_DIS
LIN {X -2.1249,Y 8.2201,Z 35,A -2.4309,B 0,C 0,E1 0.1598,E2 90.0723} C_DIS
LIN {X -1.0864,Y 8.4217,Z 35,A -2.3841,B 0,C 0,E1 0.1598,E2 90.0723} C_DIS
LIN {X -0.1899,Y 8.4884,Z 35,A -2.3481,B 0,C 0,E1 0.1598,E2 90.0724} C_DIS
LIN {X 1.0166,Y 8.4276,Z 35,A -2.3062,B 0,C 0,E1 0.1598,E2 90.0724} C_DIS
LIN {X 1.8617,Y 8.2812,Z 35,A -2.2812,B 0,C 0,E1 0.1598,E2 90.0725} C_DIS
LIN {X 2.6878,Y 8.0507,Z 35,A -2.2604,B 0,C 0,E1 0.1598,E2 90.0725} C_DIS
LIN {X 3.4865,Y 7.7383,Z 35,A -2.2442,B 0,C 0,E1 0.1598,E2 90.0725} C_DIS
Enddeposition()
END
